C09077=1065.383,91.013,-73.073,172.465,27.858,155.108
C09078=1065.389,91.262,-73.092,172.466,27.861,155.108
C09079=1065.395,91.512,-73.110,172.467,27.864,155.108
C09080=1065.401,91.761,-73.128,172.469,27.867,155.109
C09081=1065.406,92.011,-73.147,172.470,27.869,155.109
C09082=1065.413,92.260,-73.165,172.472,27.872,155.110
C09083=1065.418,92.508,-73.184,172.474,27.875,155.110
C09084=1065.424,92.758,-73.202,172.475,27.878,155.110
C09085=1065.430,93.008,-73.221,172.477,27.880,155.111
C09086=1065.436,93.257,-73.240,172.478,27.883,155.111
C09087=1065.442,93.506,-73.258,172.480,27.886,155.112
C09088=1065.447,93.755,-73.277,172.481,27.889,155.112
C09089=1065.454,94.004,-73.295,172.483,27.892,155.112
C09090=1065.460,94.288,-73.316,172.484,27.894,155.113
C09091=1065.466,94.572,-73.338,172.486,27.898,155.113
C09092=1065.473,94.855,-73.358,172.488,27.901,155.114
C09093=1065.480,95.138,-73.380,172.490,27.904,155.114
C09094=1065.486,95.389,-73.399,172.491,27.906,155.114
C09095=1065.492,95.638,-73.417,172.493,27.909,155.115
C09096=1065.498,95.886,-73.436,172.494,27.912,155.115
C09097=1065.503,96.135,-73.455,172.496,27.915,155.116
C09098=1065.510,96.385,-73.473,172.497,27.918,155.116
C09099=1065.515,96.635,-73.492,172.499,27.920,155.116
C09100=1065.521,96.883,-73.510,172.501,27.923,155.117
C09101=1065.527,97.133,-73.529,172.501,27.926,155.117
C09102=1065.533,97.382,-73.548,172.503,27.928,155.118
C09103=1065.539,97.632,-73.567,172.504,27.931,155.118
C09104=1065.545,97.881,-73.585,172.506,27.933,155.118
C09105=1065.550,98.130,-73.604,172.507,27.936,155.119
C09106=1065.557,98.379,-73.623,172.509,27.939,155.119
C09107=1065.562,98.628,-73.642,172.510,27.942,155.120
C09108=1065.569,98.877,-73.661,172.512,27.945,155.120
C09109=1065.574,99.127,-73.680,172.514,27.947,155.120
C09110=1065.580,99.376,-73.698,172.515,27.950,155.121
C09111=1065.586,99.625,-73.717,172.517,27.953,155.121
C09112=1065.592,99.874,-73.735,172.518,27.955,155.121
C09113=1065.598,100.124,-73.755,172.520,27.958,155.122
C09114=1065.604,100.373,-73.773,172.521,27.961,155.122
C09115=1065.610,100.622,-73.793,172.523,27.963,155.123
C09116=1065.616,100.871,-73.811,172.524,27.966,155.123
C09117=1065.621,101.120,-73.830,172.526,27.969,155.123
C09118=1065.628,101.369,-73.849,172.528,27.972,155.124
C09119=1065.633,101.619,-73.868,172.529,27.975,155.124
C09120=1065.639,101.868,-73.887,172.531,27.977,155.125
C09121=1065.645,102.116,-73.905,172.532,27.980,155.125
C09122=1065.651,102.366,-73.925,172.534,27.983,155.125
C09123=1065.656,102.615,-73.944,172.535,27.986,155.126
C09124=1065.663,102.864,-73.963,172.537,27.988,155.126
C09125=1065.668,103.114,-73.982,172.538,27.991,155.127
C09126=1065.673,103.363,-74.001,172.540,27.994,155.127
C09127=1065.679,103.612,-74.020,172.542,27.996,155.127
C09128=1065.686,103.861,-74.039,172.543,27.999,155.128
C09129=1065.691,104.111,-74.058,172.545,28.002,155.128
C09130=1065.697,104.360,-74.077,172.546,28.005,155.129
C09131=1065.703,104.610,-74.096,172.548,28.007,155.129
C09132=1065.709,104.859,-74.115,172.549,28.010,155.129
C09133=1065.714,105.107,-74.134,172.551,28.013,155.130
C09134=1065.720,105.357,-74.153,172.552,28.016,155.130
C09135=1065.726,105.606,-74.172,172.554,28.018,155.131
C09136=1065.732,105.855,-74.191,172.556,28.021,155.131
C09137=1065.738,106.105,-74.210,172.557,28.024,155.131
C09138=1065.744,106.354,-74.230,172.559,28.027,155.132
C09139=1065.750,106.603,-74.249,172.560,28.030,155.132
C09140=1065.756,106.852,-74.268,172.562,28.032,155.133
C09141=1065.761,107.101,-74.287,172.563,28.035,155.133
C09142=1065.767,107.350,-74.306,172.565,28.037,155.133
C09143=1065.773,107.599,-74.325,172.567,28.040,155.134
C09144=1065.779,107.849,-74.344,172.568,28.043,155.134
C09145=1065.785,108.098,-74.364,172.570,28.046,155.134
C09146=1065.790,108.347,-74.383,172.571,28.048,155.135
C09147=1065.797,108.596,-74.402,172.573,28.051,155.135
C09148=1065.802,108.846,-74.421,172.574,28.054,155.136
C09149=1065.808,109.095,-74.440,172.576,28.057,155.136
C09150=1065.814,109.344,-74.460,172.577,28.060,155.136
C09151=1065.820,109.593,-74.480,172.579,28.062,155.137
C09152=1065.826,109.842,-74.498,172.581,28.064,155.137
C09153=1065.832,110.092,-74.518,172.582,28.067,155.138
C09154=1065.838,110.376,-74.540,172.584,28.071,155.138
C09155=1065.846,110.659,-74.562,172.585,28.073,155.138
C09156=1065.852,110.943,-74.584,172.587,28.077,155.139
C09157=1065.859,111.226,-74.606,172.589,28.080,155.139
C09158=1065.865,111.476,-74.626,172.591,28.083,155.140
C09159=1065.870,111.724,-74.644,172.592,28.085,155.140
C09160=1065.875,111.974,-74.664,172.594,28.088,155.141
C09161=1065.882,112.222,-74.683,172.595,28.091,155.141
C09162=1065.888,112.472,-74.702,172.597,28.094,155.141
C09163=1065.893,112.721,-74.721,172.598,28.096,155.142
C09164=1065.899,112.970,-74.741,172.600,28.099,155.142
C09165=1065.905,113.219,-74.761,172.602,28.102,155.143
C09166=1065.911,113.468,-74.781,172.603,28.104,155.143
C09167=1065.917,113.718,-74.800,172.605,28.107,155.143
C09168=1065.922,113.967,-74.819,172.606,28.110,155.144
C09169=1065.928,114.216,-74.839,172.608,28.112,155.144
C09170=1065.934,114.465,-74.858,172.609,28.115,155.145
C09171=1065.940,114.714,-74.878,172.611,28.118,155.145
C09172=1065.946,114.964,-74.898,172.613,28.121,155.145
C09173=1065.952,115.213,-74.917,172.614,28.124,155.146
C09174=1065.957,115.462,-74.937,172.616,28.126,155.146
C09175=1065.962,115.712,-74.957,172.617,28.129,155.147
C09176=1065.968,115.960,-74.977,172.619,28.132,155.147
C09177=1065.974,116.210,-74.996,172.620,28.135,155.147
C09178=1065.980,116.459,-75.016,172.622,28.137,155.148
C09179=1065.986,116.708,-75.035,172.624,28.140,155.148
C09180=1065.992,116.957,-75.055,172.625,28.143,155.149
C09181=1065.997,117.207,-75.075,172.627,28.146,155.149
C09182=1066.003,117.455,-75.095,172.628,28.149,155.149
C09183=1066.008,117.705,-75.114,172.630,28.152,155.150
C09184=1066.014,117.954,-75.134,172.631,28.155,155.150
C09185=1066.020,118.203,-75.153,172.633,28.157,155.151
C09186=1066.026,118.452,-75.173,172.634,28.160,155.151
C09187=1066.031,118.701,-75.194,172.636,28.163,155.151
C09188=1066.037,118.950,-75.213,172.638,28.166,155.152
C09189=1066.043,119.199,-75.233,172.639,28.168,155.152
C09190=1066.049,119.449,-75.252,172.641,28.171,155.153
C09191=1066.055,119.698,-75.272,172.642,28.173,155.153
C09192=1066.060,119.947,-75.293,172.644,28.176,155.153
C09193=1066.066,120.196,-75.312,172.646,28.179,155.154
C09194=1066.072,120.445,-75.332,172.648,28.182,155.154
C09195=1066.077,120.694,-75.351,172.650,28.185,155.155
C09196=1066.083,120.943,-75.371,172.651,28.187,155.155
C09197=1066.089,121.192,-75.392,172.653,28.190,155.155
C09198=1066.095,121.442,-75.411,172.654,28.193,155.156
C09199=1066.101,121.691,-75.431,172.656,28.196,155.156
C09200=1066.107,121.940,-75.451,172.657,28.198,155.157
C09201=1066.113,122.189,-75.470,172.659,28.201,155.157
C09202=1066.118,122.439,-75.491,172.660,28.204,155.157
C09203=1066.124,122.687,-75.511,172.662,28.207,155.158
C09204=1066.130,122.937,-75.530,172.664,28.209,155.158
C09205=1066.136,123.186,-75.550,172.665,28.212,155.159
C09206=1066.142,123.434,-75.570,172.667,28.215,155.159
C09207=1066.147,123.684,-75.591,172.668,28.218,155.159
C09208=1066.153,123.934,-75.610,172.670,28.221,155.160
C09209=1066.159,124.183,-75.630,172.671,28.223,155.160
C09210=1066.165,124.431,-75.650,172.673,28.226,155.161
C09211=1066.170,124.680,-75.671,172.675,28.229,155.161
C09212=1066.176,124.930,-75.690,172.677,28.232,155.161
C09213=1066.182,125.179,-75.710,172.679,28.234,155.162
C09214=1066.188,125.428,-75.730,172.680,28.237,155.162
C09215=1066.194,125.677,-75.751,172.682,28.240,155.162
C09216=1066.200,125.926,-75.771,172.683,28.242,155.163
C09217=1066.206,126.175,-75.791,172.685,28.245,155.163
C09218=1066.212,126.459,-75.813,172.687,28.248,155.164
C09219=1066.218,126.743,-75.836,172.689,28.251,155.164
C09220=1066.226,127.026,-75.859,172.691,28.255,155.165
C09221=1066.232,127.310,-75.882,172.692,28.257,155.165
C09222=1066.238,127.559,-75.902,172.694,28.260,155.166
C09223=1066.244,127.808,-75.922,172.695,28.263,155.166
C09224=1066.249,128.057,-75.942,172.698,28.266,155.166
C09225=1066.256,128.306,-75.962,172.699,28.269,155.167
C09226=1066.262,128.555,-75.982,172.701,28.271,155.167
C09227=1066.267,128.804,-76.003,172.703,28.274,155.167
C09228=1066.273,129.053,-76.023,172.704,28.276,155.168
C09229=1066.280,129.303,-76.043,172.706,28.279,155.168
C09230=1066.286,129.551,-76.063,172.707,28.282,155.169
C09231=1066.291,129.800,-76.084,172.709,28.285,155.169
C09232=1066.297,130.050,-76.103,172.710,28.287,155.169
C09233=1066.303,130.299,-76.123,172.712,28.290,155.170
C09234=1066.309,130.549,-76.144,172.714,28.292,155.170
C09235=1066.315,130.797,-76.164,172.716,28.295,155.171
C09236=1066.321,131.046,-76.184,172.718,28.298,155.171
C09237=1066.327,131.296,-76.205,172.719,28.301,155.171
C09238=1066.333,131.545,-76.225,172.721,28.304,155.172
C09239=1066.339,131.794,-76.245,172.723,28.306,155.172
C09240=1066.344,132.043,-76.266,172.724,28.309,155.173
C09241=1066.351,132.292,-76.286,172.726,28.312,155.173
C09242=1066.356,132.541,-76.307,172.727,28.315,155.173
C09243=1066.362,132.790,-76.327,172.729,28.317,155.174
C09244=1066.367,133.039,-76.347,172.730,28.320,155.174
C09245=1066.374,133.288,-76.368,172.733,28.323,155.175
C09246=1066.379,133.537,-76.388,172.735,28.326,155.175
C09247=1066.384,133.786,-76.409,172.736,28.329,155.175
C09248=1066.390,134.035,-76.429,172.738,28.331,155.176
C09249=1066.396,134.285,-76.450,172.739,28.334,155.176
C09250=1066.402,134.534,-76.470,172.741,28.337,155.177
C09251=1066.408,134.782,-76.491,172.742,28.340,155.177
C09252=1066.414,135.031,-76.511,172.744,28.342,155.177
C09253=1066.420,135.281,-76.532,172.746,28.345,155.178
C09254=1066.425,135.530,-76.552,172.747,28.348,155.178
C09255=1066.431,135.779,-76.572,172.750,28.350,155.178
C09256=1066.437,136.029,-76.593,172.751,28.353,155.179
C09257=1066.443,136.277,-76.614,172.753,28.356,155.179
C09258=1066.448,136.526,-76.634,172.755,28.359,155.180
C09259=1066.454,136.776,-76.655,172.756,28.361,155.180
C09260=1066.460,137.025,-76.675,172.758,28.364,155.180
C09261=1066.466,137.273,-76.697,172.759,28.367,155.181
C09262=1066.472,137.523,-76.717,172.761,28.370,155.181
C09263=1066.477,137.772,-76.737,172.763,28.373,155.182
C09264=1066.483,138.021,-76.758,172.765,28.375,155.182
C09265=1066.490,138.270,-76.779,172.767,28.378,155.182
C09266=1066.495,138.519,-76.800,172.768,28.381,155.183
C09267=1066.500,138.768,-76.820,172.770,28.384,155.183
C09268=1066.507,139.018,-76.840,172.771,28.386,155.184
C09269=1066.512,139.266,-76.862,172.773,28.389,155.184
C09270=1066.518,139.515,-76.882,172.775,28.392,155.184
C09271=1066.524,139.765,-76.903,172.777,28.395,155.185
C09272=1066.530,140.013,-76.924,172.779,28.398,155.185
C09273=1066.535,140.262,-76.944,172.780,28.400,155.186
C09274=1066.542,140.512,-76.965,172.782,28.403,155.186
C09275=1066.547,140.760,-76.986,172.783,28.406,155.187
C09276=1066.552,141.010,-77.007,172.785,28.409,155.187
C09277=1066.559,141.259,-77.028,172.788,28.411,155.187
C09278=1066.564,141.508,-77.049,172.789,28.414,155.188
C09279=1066.570,141.757,-77.069,172.791,28.417,155.188
C09280=1066.576,142.006,-77.090,172.792,28.420,155.189
C09281=1066.581,142.255,-77.111,172.794,28.422,155.189
C09282=1066.588,142.539,-77.135,172.796,28.426,155.189
C09283=1066.594,142.822,-77.159,172.798,28.429,155.190
C09284=1066.600,143.105,-77.183,172.799,28.432,155.190
C09285=1066.608,143.389,-77.206,172.802,28.435,155.191
C09286=1066.613,143.638,-77.227,172.804,28.438,155.191
C09287=1066.619,143.887,-77.249,172.805,28.441,155.192
C09288=1066.625,144.136,-77.269,172.807,28.443,155.192
C09289=1066.630,144.385,-77.290,172.809,28.446,155.192
C09290=1066.636,144.635,-77.311,172.811,28.449,155.193
C09291=1066.642,144.883,-77.332,172.812,28.452,155.193
C09292=1066.648,145.132,-77.354,172.814,28.454,155.194
C09293=1066.654,145.381,-77.374,172.816,28.457,155.194
C09294=1066.660,145.630,-77.396,172.817,28.460,155.194
C09295=1066.665,145.880,-77.416,172.820,28.463,155.195
C09296=1066.671,146.128,-77.438,172.821,28.466,155.195
C09297=1066.677,146.378,-77.458,172.823,28.468,155.196
C09298=1066.683,146.626,-77.479,172.825,28.471,155.196
C09299=1066.689,146.875,-77.501,172.826,28.474,155.196
C09300=1066.694,147.124,-77.521,172.828,28.477,155.197
C09301=1066.700,147.374,-77.543,172.830,28.480,155.197
C09302=1066.706,147.623,-77.564,172.832,28.482,155.198
C09303=1066.712,147.872,-77.585,172.833,28.485,155.198
C09304=1066.717,148.120,-77.606,172.835,28.488,155.198
C09305=1066.723,148.370,-77.627,172.837,28.491,155.199
C09306=1066.729,148.619,-77.649,172.839,28.494,155.199
C09307=1066.735,148.868,-77.670,172.841,28.496,155.200
C09308=1066.740,149.117,-77.691,172.842,28.499,155.200
C09309=1066.746,149.366,-77.712,172.844,28.502,155.200
C09310=1066.752,149.615,-77.734,172.846,28.504,155.201
C09311=1066.758,149.864,-77.755,172.847,28.507,155.201
C09312=1066.763,150.113,-77.776,172.850,28.510,155.202
C09313=1066.769,150.362,-77.797,172.851,28.513,155.202
C09314=1066.775,150.611,-77.819,172.853,28.516,155.202
C09315=1066.780,150.860,-77.839,172.855,28.518,155.203
C09316=1066.787,151.109,-77.861,172.856,28.521,155.203
C09317=1066.792,151.358,-77.882,172.859,28.524,155.204
C09318=1066.798,151.607,-77.904,172.860,28.527,155.204
C09319=1066.804,151.856,-77.926,172.862,28.530,155.204
C09320=1066.809,152.106,-77.947,172.863,28.532,155.205
C09321=1066.815,152.355,-77.968,172.866,28.536,155.205
C09322=1066.821,152.603,-77.990,172.868,28.539,155.206
C09323=1066.827,152.852,-78.011,172.869,28.541,155.206
C09324=1066.832,153.101,-78.033,172.871,28.544,155.207
C09325=1066.839,153.350,-78.054,172.872,28.547,155.207
C09326=1066.844,153.599,-78.075,172.875,28.550,155.207
C09327=1066.850,153.848,-78.096,172.876,28.552,155.208
C09328=1066.856,154.097,-78.118,172.878,28.555,155.208
C09329=1066.861,154.346,-78.140,172.880,28.558,155.209
C09330=1066.867,154.596,-78.161,172.881,28.561,155.209
C09331=1066.873,154.844,-78.183,172.884,28.564,155.209
C09332=1066.879,155.093,-78.204,172.885,28.566,155.210
C09333=1066.884,155.342,-78.226,172.887,28.569,155.210
C09334=1066.891,155.591,-78.247,172.889,28.572,155.211
C09335=1066.895,155.840,-78.269,172.891,28.575,155.211
C09336=1066.902,156.089,-78.291,172.893,28.578,155.211
C09337=1066.908,156.338,-78.312,172.894,28.580,155.212
C09338=1066.913,156.587,-78.334,172.896,28.583,155.212
C09339=1066.919,156.836,-78.356,172.899,28.586,155.213
C09340=1066.924,157.085,-78.377,172.900,28.589,155.213
C09341=1066.930,157.334,-78.399,172.902,28.591,155.213
C09342=1066.937,157.583,-78.420,172.903,28.594,155.214
C09343=1066.941,157.832,-78.442,172.906,28.598,155.214
C09344=1066.948,158.081,-78.464,172.907,28.600,155.215
C09345=1066.953,158.330,-78.485,172.909,28.603,155.215
C09346=1066.960,158.613,-78.510,172.912,28.606,155.215
C09347=1066.966,158.896,-78.535,172.913,28.609,155.216
C09348=1066.973,159.180,-78.560,172.916,28.612,155.216
C09349=1066.980,159.463,-78.584,172.917,28.616,155.217
C09350=1066.985,159.712,-78.606,172.920,28.619,155.217
C09351=1066.991,159.961,-78.628,172.921,28.621,155.218
C09352=1066.996,160.210,-78.649,172.923,28.624,155.218
C09353=1067.003,160.459,-78.671,172.925,28.627,155.219
C09354=1067.008,160.708,-78.693,172.927,28.630,155.219
C09355=1067.015,160.957,-78.715,172.929,28.632,155.219
C09356=1067.020,161.205,-78.737,172.930,28.635,155.220
C09357=1067.026,161.455,-78.759,172.932,28.638,155.220
C09358=1067.031,161.703,-78.780,172.935,28.641,155.221
C09359=1067.036,161.953,-78.802,172.936,28.644,155.221
C09360=1067.042,162.202,-78.825,172.938,28.647,155.221
C09361=1067.048,162.450,-78.847,172.939,28.650,155.222
C09362=1067.053,162.700,-78.869,172.942,28.653,155.222
C09363=1067.059,162.948,-78.890,172.943,28.656,155.223
C09364=1067.065,163.197,-78.913,172.945,28.659,155.223
C09365=1067.070,163.447,-78.935,172.948,28.662,155.224
C09366=1067.075,163.695,-78.956,172.949,28.665,155.224
C09367=1067.081,163.945,-78.979,172.951,28.668,155.224
C09368=1067.087,164.193,-79.001,172.952,28.670,155.225
C09369=1067.092,164.442,-79.023,172.955,28.673,155.225
C09370=1067.098,164.692,-79.045,172.956,28.677,155.226
C09371=1067.103,164.940,-79.067,172.958,28.679,155.226
C09372=1067.109,165.189,-79.089,172.961,28.682,155.227
C09373=1067.114,165.439,-79.112,172.962,28.685,155.227
C09374=1067.120,165.687,-79.134,172.964,28.688,155.227
C09375=1067.126,165.936,-79.156,172.965,28.691,155.228
C09376=1067.131,166.186,-79.178,172.968,28.694,155.228
C09377=1067.138,166.434,-79.200,172.970,28.697,155.229
C09378=1067.142,166.683,-79.222,172.971,28.699,155.229
C09379=1067.148,166.932,-79.245,172.974,28.702,155.230
C09380=1067.154,167.181,-79.267,172.975,28.706,155.230
C09381=1067.159,167.429,-79.289,172.977,28.708,155.230
C09382=1067.165,167.679,-79.312,172.979,28.711,155.231
C09383=1067.171,167.928,-79.333,172.981,28.714,155.231
C09384=1067.177,168.177,-79.356,172.983,28.717,155.232
C09385=1067.182,168.426,-79.378,172.984,28.720,155.232
C09386=1067.188,168.674,-79.400,172.987,28.723,155.233
C09387=1067.193,168.924,-79.423,172.988,28.726,155.233
C09388=1067.199,169.172,-79.445,172.990,28.728,155.233
C09389=1067.205,169.421,-79.467,172.993,28.731,155.234
C09390=1067.210,169.670,-79.490,172.994,28.735,155.234
C09391=1067.216,169.920,-79.512,172.996,28.737,155.235
C09392=1067.222,170.168,-79.534,172.998,28.740,155.235
C09393=1067.227,170.417,-79.556,173.000,28.743,155.236
C09394=1067.233,170.666,-79.579,173.002,28.746,155.236
C09395=1067.239,170.915,-79.602,173.004,28.749,155.236
C09396=1067.245,171.164,-79.624,173.006,28.752,155.237
C09397=1067.251,171.413,-79.647,173.007,28.755,155.237
C09398=1067.255,171.662,-79.669,173.010,28.758,155.238
C09399=1067.262,171.910,-79.691,173.012,28.760,155.238
C09400=1067.268,172.159,-79.714,173.013,28.763,155.238
C09401=1067.273,172.409,-79.736,173.016,28.766,155.239
C09402=1067.279,172.658,-79.759,173.017,28.769,155.239
C09403=1067.285,172.906,-79.781,173.019,28.772,155.240
C09404=1067.290,173.155,-79.803,173.021,28.775,155.240
C09405=1067.296,173.404,-79.826,173.023,28.778,155.241
C09406=1067.301,173.653,-79.849,173.025,28.780,155.241
C09407=1067.308,173.902,-79.871,173.027,28.784,155.242
C09408=1067.313,174.151,-79.894,173.029,28.786,155.242
C09409=1067.319,174.400,-79.917,173.031,28.789,155.242
C09410=1067.325,174.683,-79.941,173.033,28.793,155.243
C09411=1067.332,174.966,-79.967,173.036,28.796,155.243
C09412=1067.338,175.248,-79.993,173.038,28.799,155.244
C09413=1067.345,175.531,-80.019,173.040,28.802,155.244
C09414=1067.351,175.780,-80.041,173.042,28.805,155.245
C09415=1067.357,176.029,-80.064,173.044,28.808,155.245
C09416=1067.363,176.278,-80.087,173.045,28.811,155.245
C09417=1067.368,176.527,-80.109,173.048,28.814,155.246
C09418=1067.374,176.776,-80.132,173.050,28.817,155.246
C09419=1067.380,177.025,-80.155,173.052,28.820,155.247
C09420=1067.386,177.273,-80.178,173.054,28.823,155.247
C09421=1067.392,177.522,-80.200,173.055,28.825,155.248
C09422=1067.397,177.772,-80.223,173.058,28.828,155.248
C09423=1067.403,178.020,-80.245,173.060,28.831,155.248
C09424=1067.409,178.269,-80.268,173.062,28.835,155.249
C09425=1067.414,178.518,-80.291,173.064,28.837,155.249
C09426=1067.420,178.766,-80.313,173.065,28.840,155.250
C09427=1067.426,179.015,-80.336,173.068,28.843,155.250
C09428=1067.432,179.264,-80.359,173.070,28.846,155.251
C09429=1067.438,179.513,-80.382,173.072,28.849,155.251
C09430=1067.444,179.762,-80.405,173.074,28.851,155.251
C09431=1067.450,180.011,-80.428,173.075,28.854,155.252
C09432=1067.455,180.260,-80.450,173.078,28.857,155.252
C09433=1067.461,180.509,-80.473,173.080,28.860,155.253
C09434=1067.467,180.758,-80.495,173.082,28.863,155.253
C09435=1067.473,181.006,-80.518,173.084,28.866,155.253
C09436=1067.479,181.256,-80.541,173.086,28.869,155.254
C09437=1067.485,181.505,-80.564,173.088,28.871,155.254
C09438=1067.491,181.754,-80.587,173.090,28.875,155.255
C09439=1067.496,182.003,-80.610,173.092,28.878,155.255
C09440=1067.503,182.251,-80.633,173.094,28.880,155.256
C09441=1067.509,182.500,-80.656,173.096,28.883,155.256
C09442=1067.514,182.749,-80.678,173.098,28.886,155.256
C09443=1067.520,182.997,-80.702,173.101,28.889,155.257
C09444=1067.526,183.246,-80.725,173.102,28.892,155.257
C09445=1067.532,183.495,-80.748,173.104,28.894,155.258
C09446=1067.538,183.744,-80.771,173.106,28.898,155.258
C09447=1067.544,183.993,-80.793,173.108,28.900,155.258
C09448=1067.550,184.242,-80.816,173.111,28.903,155.259
C09449=1067.556,184.491,-80.840,173.112,28.906,155.259
C09450=1067.562,184.740,-80.863,173.115,28.909,155.260
C09451=1067.568,184.989,-80.885,173.116,28.912,155.260
C09452=1067.573,185.238,-80.910,173.119,28.915,155.261
C09453=1067.579,185.486,-80.933,173.121,28.918,155.261
C09454=1067.584,185.735,-80.956,173.122,28.921,155.262
C09455=1067.589,185.985,-80.979,173.125,28.924,155.262
C09456=1067.595,186.233,-81.002,173.126,28.927,155.262
C09457=1067.601,186.482,-81.026,173.129,28.930,155.263
C09458=1067.606,186.731,-81.049,173.130,28.933,155.263
C09459=1067.612,186.980,-81.072,173.133,28.936,155.264
C09460=1067.618,187.229,-81.095,173.135,28.939,155.264
C09461=1067.623,187.477,-81.119,173.137,28.943,155.265
C09462=1067.629,187.726,-81.142,173.139,28.945,155.265
C09463=1067.634,187.975,-81.165,173.141,28.949,155.266
C09464=1067.640,188.224,-81.190,173.143,28.952,155.266
C09465=1067.645,188.473,-81.213,173.146,28.954,155.266
C09466=1067.651,188.722,-81.236,173.147,28.958,155.267
C09467=1067.656,188.970,-81.260,173.149,28.960,155.267
C09468=1067.662,189.219,-81.283,173.151,28.964,155.268
C09469=1067.668,189.468,-81.306,173.153,28.967,155.268
C09470=1067.673,189.716,-81.330,173.156,28.970,155.269
C09471=1067.679,189.965,-81.353,173.157,28.973,155.269
C09472=1067.685,190.215,-81.376,173.160,28.976,155.270
C09473=1067.691,190.464,-81.400,173.161,28.979,155.270
C09474=1067.697,190.745,-81.427,173.164,28.982,155.271
C09475=1067.704,191.028,-81.454,173.166,28.986,155.271
C09476=1067.710,191.311,-81.480,173.169,28.989,155.272
C09477=1067.716,191.593,-81.507,173.171,28.993,155.272
C09478=1067.722,191.841,-81.530,173.173,28.996,155.273
C09479=1067.728,192.091,-81.554,173.176,28.998,155.273
C09480=1067.734,192.340,-81.578,173.177,29.002,155.273
C09481=1067.739,192.588,-81.601,173.180,29.005,155.274
C09482=1067.745,192.837,-81.625,173.181,29.008,155.274
C09483=1067.750,193.086,-81.648,173.184,29.011,155.275
C09484=1067.756,193.334,-81.672,173.186,29.014,155.275
C09485=1067.762,193.584,-81.696,173.188,29.017,155.276
C09486=1067.768,193.832,-81.719,173.190,29.020,155.276
C09487=1067.773,194.081,-81.743,173.192,29.023,155.277
C09488=1067.779,194.330,-81.766,173.194,29.026,155.277
C09489=1067.784,194.578,-81.791,173.196,29.029,155.278
C09490=1067.791,194.828,-81.814,173.198,29.032,155.278
C09491=1067.797,195.076,-81.838,173.201,29.035,155.278
C09492=1067.802,195.325,-81.862,173.202,29.038,155.279
C09493=1067.808,195.574,-81.885,173.205,29.041,155.279
C09494=1067.814,195.823,-81.909,173.207,29.045,155.280
C09495=1067.819,196.072,-81.932,173.209,29.047,155.280
C09496=1067.825,196.321,-81.957,173.212,29.050,155.281
C09497=1067.831,196.569,-81.980,173.213,29.053,155.281
C09498=1067.837,196.818,-82.004,173.216,29.056,155.281
C09499=1067.842,197.067,-82.028,173.217,29.060,155.282
C09500=1067.848,197.315,-82.052,173.220,29.062,155.282
C09501=1067.854,197.564,-82.076,173.222,29.066,155.283
C09502=1067.860,197.813,-82.099,173.224,29.069,155.283
C09503=1067.865,198.062,-82.123,173.227,29.072,155.284
C09504=1067.871,198.310,-82.147,173.228,29.075,155.284
C09505=1067.877,198.560,-82.172,173.231,29.078,155.285
C09506=1067.883,198.809,-82.195,173.233,29.081,155.285
C09507=1067.888,199.057,-82.219,173.235,29.084,155.286
C09508=1067.895,199.306,-82.243,173.237,29.087,155.286
C09509=1067.901,199.554,-82.267,173.239,29.090,155.287
C09510=1067.906,199.803,-82.291,173.242,29.093,155.287
C09511=1067.913,200.053,-82.314,173.244,29.096,155.287
C09512=1067.918,200.301,-82.338,173.246,29.099,155.288
C09513=1067.924,200.549,-82.362,173.248,29.102,155.288
C09514=1067.930,200.799,-82.387,173.250,29.105,155.289
C09515=1067.936,201.047,-82.410,173.252,29.108,155.289
C09516=1067.941,201.296,-82.435,173.255,29.111,155.290
C09517=1067.948,201.545,-82.459,173.257,29.114,155.290
C09518=1067.953,201.794,-82.482,173.259,29.118,155.291
C09519=1067.959,202.043,-82.506,173.261,29.120,155.291
C09520=1067.965,202.291,-82.530,173.263,29.124,155.292
C09521=1067.970,202.540,-82.555,173.266,29.127,155.292
C09522=1067.977,202.789,-82.579,173.268,29.130,155.292
C09523=1067.982,203.037,-82.603,173.270,29.133,155.293
C09524=1067.987,203.286,-82.627,173.272,29.136,155.293
C09525=1067.993,203.535,-82.652,173.274,29.139,155.294
C09526=1067.998,203.784,-82.676,173.277,29.142,155.294
C09527=1068.004,204.032,-82.700,173.279,29.146,155.295
C09528=1068.010,204.282,-82.724,173.281,29.148,155.295
C09529=1068.016,204.530,-82.749,173.283,29.152,155.296
C09530=1068.022,204.779,-82.773,173.286,29.155,155.296
C09531=1068.028,205.028,-82.797,173.287,29.158,155.297
C09532=1068.033,205.276,-82.821,173.290,29.162,155.297
C09533=1068.039,205.525,-82.846,173.292,29.164,155.298
C09534=1068.044,205.773,-82.871,173.294,29.168,155.298
C09535=1068.050,206.023,-82.895,173.297,29.171,155.299
C09536=1068.056,206.271,-82.919,173.298,29.174,155.299
C09537=1068.062,206.520,-82.943,173.301,29.177,155.300
C09538=1068.086,207.564,-83.046,173.447,29.251,155.303
C09539=1068.092,207.797,-83.070,173.450,29.255,155.304
C09540=1068.097,208.030,-83.093,173.451,29.259,155.305
C09541=1068.103,208.263,-83.117,173.453,29.263,155.305
C09542=1068.108,208.496,-83.140,173.455,29.267,155.306
C09543=1068.114,208.728,-83.164,173.457,29.270,155.307
C09544=1068.119,208.962,-83.188,173.458,29.274,155.307
C09545=1068.125,209.194,-83.211,173.461,29.278,155.308
C09546=1068.130,209.427,-83.234,173.462,29.282,155.308
C09547=1068.136,209.676,-83.260,173.465,29.286,155.309
C09548=1068.142,209.924,-83.285,173.466,29.290,155.310
C09549=1068.148,210.173,-83.311,173.469,29.294,155.311
C09550=1068.155,210.422,-83.336,173.470,29.298,155.311
C09551=1068.160,210.670,-83.360,173.473,29.302,155.312
C09552=1068.166,210.919,-83.386,173.474,29.306,155.313
C09553=1068.171,211.168,-83.412,173.477,29.310,155.313
C09554=1068.178,211.417,-83.437,173.478,29.314,155.314
C09555=1068.184,211.665,-83.462,173.481,29.319,155.315
C09556=1068.189,211.913,-83.487,173.482,29.322,155.315
C09557=1068.195,212.162,-83.513,173.485,29.326,155.316
C09558=1068.201,212.411,-83.538,173.486,29.331,155.317
C09559=1068.207,212.660,-83.564,173.489,29.335,155.317
C09560=1068.214,212.908,-83.589,173.490,29.338,155.318
C09561=1068.219,213.157,-83.615,173.493,29.342,155.319
C09562=1068.225,213.405,-83.640,173.494,29.347,155.319
C09563=1068.231,213.654,-83.665,173.497,29.351,155.320
C09564=1068.236,213.903,-83.691,173.499,29.354,155.321
C09565=1068.243,214.152,-83.717,173.501,29.359,155.322
C09566=1068.249,214.400,-83.742,173.503,29.363,155.322
C09567=1068.254,214.649,-83.768,173.505,29.367,155.323
C09568=1068.260,214.898,-83.793,173.507,29.371,155.324
C09569=1068.266,215.146,-83.820,173.509,29.375,155.324
C09570=1068.272,215.394,-83.845,173.511,29.379,155.325
C09571=1068.278,215.643,-83.870,173.513,29.383,155.326
C09572=1068.283,215.892,-83.896,173.516,29.387,155.326
C09573=1068.290,216.141,-83.921,173.517,29.391,155.327
C09574=1068.295,216.390,-83.947,173.520,29.396,155.328
C09575=1068.301,216.638,-83.973,173.521,29.399,155.328
C09576=1068.308,216.886,-83.999,173.524,29.403,155.329
C09577=1068.313,217.135,-84.025,173.525,29.407,155.330
C09578=1068.319,217.383,-84.050,173.528,29.412,155.330
C09579=1068.324,217.616,-84.074,173.529,29.415,155.331
C09580=1068.330,217.847,-84.098,173.532,29.419,155.332
C09581=1068.335,218.080,-84.122,173.533,29.423,155.332
C09582=1068.341,218.311,-84.146,173.535,29.426,155.333
C09583=1068.347,218.543,-84.170,173.537,29.430,155.334
C09584=1068.352,218.776,-84.194,173.539,29.434,155.334
C09585=1068.358,219.007,-84.218,173.542,29.437,155.335
C09586=1068.363,219.239,-84.242,173.543,29.441,155.335
C09587=1068.370,219.487,-84.269,173.545,29.445,155.336
C09588=1068.375,219.736,-84.294,173.547,29.449,155.337
C09589=1068.381,219.985,-84.320,173.550,29.453,155.337
C09590=1068.388,220.233,-84.346,173.551,29.457,155.338
C09591=1068.393,220.482,-84.372,173.554,29.461,155.339
C09592=1068.399,220.730,-84.397,173.555,29.466,155.340
C09593=1068.405,220.979,-84.424,173.558,29.469,155.340
C09594=1068.411,221.227,-84.449,173.560,29.473,155.341
C09595=1068.416,221.446,-84.472,173.562,29.477,155.341
C09596=1068.422,221.664,-84.495,173.563,29.480,155.342
C09597=1068.427,221.883,-84.518,173.565,29.484,155.343
C09598=1068.432,222.101,-84.541,173.568,29.488,155.343
C09599=1068.437,222.320,-84.563,173.569,29.491,155.344
C09600=1068.442,222.539,-84.586,173.571,29.495,155.344
C09601=1068.447,222.756,-84.609,173.572,29.498,155.345
C09602=1068.452,222.974,-84.632,173.575,29.502,155.346
C09603=1068.458,223.223,-84.658,173.577,29.505,155.346
C09604=1068.464,223.472,-84.684,173.579,29.510,155.347
C09605=1068.469,223.720,-84.711,173.581,29.514,155.348
C09606=1068.476,223.970,-84.737,173.583,29.518,155.348
C09607=1068.482,224.218,-84.763,173.586,29.522,155.349
C09608=1068.488,224.466,-84.790,173.587,29.526,155.350
C09609=1068.494,224.715,-84.815,173.590,29.530,155.350
C09610=1068.500,224.963,-84.842,173.591,29.534,155.351
C09611=1068.505,225.212,-84.868,173.594,29.538,155.352
C09612=1068.512,225.460,-84.894,173.596,29.542,155.352
C09613=1068.517,225.709,-84.921,173.598,29.546,155.353
C09614=1068.523,225.958,-84.947,173.600,29.550,155.354
C09615=1068.529,226.206,-84.973,173.602,29.554,155.354
C09616=1068.535,226.455,-84.999,173.605,29.558,155.355
C09617=1068.541,226.703,-85.025,173.607,29.562,155.356
C09618=1068.546,226.951,-85.052,173.609,29.566,155.357
C09619=1068.553,227.200,-85.079,173.611,29.570,155.357
C09620=1068.559,227.449,-85.104,173.614,29.574,155.358
C09621=1068.565,227.698,-85.131,173.615,29.577,155.358
C09622=1068.571,227.946,-85.157,173.618,29.582,155.359
C09623=1068.576,228.195,-85.183,173.620,29.586,155.360
C09624=1068.583,228.443,-85.209,173.622,29.590,155.361
C09625=1068.589,228.692,-85.236,173.624,29.594,155.361
C09626=1068.595,228.940,-85.263,173.626,29.597,155.362
C09627=1068.601,229.189,-85.290,173.628,29.601,155.362
C09628=1068.607,229.437,-85.315,173.631,29.605,155.363
C09629=1068.612,229.686,-85.342,173.633,29.610,155.364
C09630=1068.619,229.935,-85.369,173.635,29.614,155.365
C09631=1068.625,230.183,-85.395,173.638,29.617,155.365
C09632=1068.630,230.431,-85.422,173.639,29.621,155.366
C09633=1068.636,230.680,-85.449,173.642,29.625,155.366
C09634=1068.642,230.929,-85.475,173.644,29.630,155.367
C09635=1068.647,231.177,-85.501,173.646,29.633,155.368
C09636=1068.654,231.426,-85.528,173.648,29.637,155.369
C09637=1068.660,231.675,-85.555,173.651,29.641,155.369
C09638=1068.665,231.923,-85.582,173.652,29.646,155.370
C09639=1068.671,232.171,-85.608,173.655,29.650,155.371
C09640=1068.677,232.420,-85.635,173.658,29.653,155.371
C09641=1068.683,232.669,-85.662,173.659,29.657,155.372
C09642=1068.689,232.917,-85.689,173.662,29.661,155.373
C09643=1068.695,233.165,-85.715,173.664,29.666,155.373
C09644=1068.701,233.414,-85.742,173.666,29.669,155.374
C09645=1068.706,233.662,-85.768,173.668,29.673,155.375
C09646=1068.713,233.911,-85.796,173.671,29.677,155.375
C09647=1068.719,234.160,-85.822,173.673,29.681,155.376
C09648=1068.724,234.408,-85.849,173.675,29.686,155.377
C09649=1068.730,234.656,-85.875,173.678,29.689,155.377
C09650=1068.736,234.905,-85.902,173.679,29.693,155.378
C09651=1068.741,235.120,-85.926,173.682,29.697,155.379
C09652=1068.746,235.334,-85.950,173.683,29.700,155.379
C09653=1068.752,235.548,-85.972,173.685,29.703,155.380
C09654=1068.757,235.762,-85.995,173.687,29.707,155.380
C09655=1068.761,235.976,-86.019,173.689,29.711,155.381
C09656=1068.766,236.191,-86.042,173.691,29.714,155.382
C09657=1068.772,236.405,-86.065,173.692,29.718,155.382
C09658=1068.777,236.620,-86.089,173.695,29.721,155.383
C09659=1068.783,236.868,-86.115,173.697,29.725,155.383
C09660=1068.789,237.117,-86.142,173.699,29.729,155.384
C09661=1068.795,237.365,-86.169,173.702,29.733,155.385
C09662=1068.800,237.614,-86.197,173.704,29.737,155.385
C09663=1068.806,237.862,-86.224,173.706,29.741,155.386
C09664=1068.812,238.110,-86.250,173.708,29.745,155.387
C09665=1068.818,238.359,-86.277,173.711,29.749,155.387
C09666=1068.824,238.607,-86.305,173.713,29.752,155.388
C09667=1068.830,238.856,-86.331,173.715,29.757,155.389
C09668=1068.836,239.105,-86.359,173.718,29.761,155.389
C09669=1068.842,239.353,-86.386,173.720,29.765,155.390
C09670=1068.848,239.602,-86.413,173.722,29.768,155.391
C09671=1068.854,239.850,-86.440,173.724,29.772,155.391
C09672=1068.860,240.098,-86.467,173.727,29.776,155.392
C09673=1068.866,240.347,-86.495,173.729,29.780,155.393
C09674=1068.872,240.596,-86.522,173.731,29.784,155.393
C09675=1068.878,240.843,-86.549,173.734,29.788,155.394
C09676=1068.884,241.092,-86.576,173.736,29.792,155.395
C09677=1068.889,241.340,-86.604,173.738,29.796,155.395
C09678=1068.896,241.590,-86.631,173.740,29.800,155.396
C09679=1068.902,241.837,-86.658,173.743,29.804,155.397
C09680=1068.908,242.086,-86.685,173.746,29.808,155.397
C09681=1068.913,242.335,-86.713,173.747,29.812,155.398
C09682=1068.919,242.583,-86.740,173.750,29.816,155.399
C09683=1068.926,242.832,-86.767,173.752,29.820,155.399
C09684=1068.931,243.080,-86.795,173.755,29.824,155.400
C09685=1068.938,243.328,-86.823,173.756,29.828,155.401
C09686=1068.943,243.577,-86.850,173.759,29.832,155.402
C09687=1068.949,243.825,-86.877,173.762,29.836,155.402
C09688=1068.954,244.074,-86.905,173.764,29.840,155.403
C09689=1068.961,244.322,-86.932,173.766,29.844,155.404
C09690=1068.967,244.571,-86.959,173.768,29.848,155.404
C09691=1068.972,244.819,-86.987,173.771,29.852,155.405
C09692=1068.979,245.067,-87.015,173.773,29.856,155.406
C09693=1068.984,245.316,-87.042,173.775,29.860,155.406
C09694=1068.990,245.564,-87.070,173.778,29.864,155.407
C09695=1068.996,245.813,-87.098,173.780,29.868,155.408
C09696=1069.002,246.061,-87.124,173.783,29.872,155.408
C09697=1069.008,246.310,-87.153,173.784,29.876,155.409
C09698=1069.014,246.557,-87.180,173.787,29.880,155.410
C09699=1069.019,246.807,-87.208,173.790,29.884,155.410
C09700=1069.026,247.054,-87.235,173.792,29.888,155.411
C09701=1069.031,247.303,-87.263,173.794,29.892,155.412
C09702=1069.037,247.551,-87.291,173.796,29.896,155.412
C09703=1069.043,247.800,-87.318,173.799,29.900,155.413
C09704=1069.049,248.048,-87.346,173.801,29.904,155.414
C09705=1069.054,248.297,-87.375,173.804,29.908,155.414
C09706=1069.061,248.545,-87.402,173.806,29.912,155.415
C09707=1069.065,248.756,-87.426,173.808,29.916,155.416
C09708=1069.070,248.967,-87.450,173.810,29.919,155.416
C09709=1069.075,249.179,-87.474,173.812,29.922,155.417
C09710=1069.080,249.390,-87.497,173.814,29.926,155.417
C09711=1069.085,249.601,-87.521,173.816,29.929,155.418
C09712=1069.090,249.812,-87.545,173.818,29.932,155.419
C09713=1069.095,250.023,-87.568,173.820,29.936,155.419
C09714=1069.100,250.234,-87.592,173.822,29.939,155.420
C09715=1069.106,250.482,-87.620,173.824,29.943,155.420
C09716=1069.112,250.731,-87.648,173.827,29.947,155.421
C09717=1069.118,250.979,-87.676,173.829,29.951,155.422
C09718=1069.124,251.228,-87.704,173.832,29.955,155.422
C09719=1069.129,251.476,-87.732,173.834,29.959,155.423
C09720=1069.135,251.724,-87.760,173.836,29.963,155.424
C09721=1069.141,251.972,-87.788,173.839,29.967,155.425
C09722=1069.147,252.221,-87.816,173.841,29.971,155.425
C09723=1069.152,252.469,-87.844,173.844,29.975,155.426
C09724=1069.158,252.718,-87.872,173.846,29.979,155.427
C09725=1069.165,252.966,-87.900,173.848,29.983,155.427
C09726=1069.170,253.214,-87.928,173.851,29.987,155.428
C09727=1069.176,253.463,-87.956,173.853,29.991,155.429
C09728=1069.182,253.711,-87.984,173.856,29.995,155.429
C09729=1069.188,253.959,-88.012,173.859,29.999,155.430
C09730=1069.194,254.208,-88.040,173.860,30.003,155.431
C09731=1069.200,254.456,-88.068,173.863,30.007,155.431
C09732=1069.206,254.704,-88.097,173.865,30.011,155.432
C09733=1069.212,254.953,-88.126,173.868,30.015,155.433
C09734=1069.218,255.201,-88.153,173.871,30.019,155.433
C09735=1069.224,255.450,-88.181,173.873,30.023,155.434
C09736=1069.230,255.698,-88.210,173.875,30.027,155.435
C09737=1069.235,255.946,-88.238,173.877,30.031,155.435
C09738=1069.241,256.195,-88.267,173.880,30.035,155.436
C09739=1069.248,256.443,-88.294,173.883,30.039,155.437
C09740=1069.254,256.692,-88.323,173.885,30.043,155.437
C09741=1069.259,256.940,-88.351,173.888,30.046,155.438
C09742=1069.266,257.188,-88.380,173.890,30.051,155.439
C09743=1069.271,257.437,-88.408,173.892,30.055,155.439
C09744=1069.277,257.685,-88.436,173.895,30.058,155.440
C09745=1069.284,257.933,-88.464,173.897,30.062,155.441
C09746=1069.290,258.181,-88.493,173.900,30.066,155.441
C09747=1069.296,258.430,-88.521,173.902,30.070,155.442
C09748=1069.301,258.678,-88.550,173.905,30.075,155.443
C09749=1069.307,258.926,-88.578,173.908,30.079,155.443
C09750=1069.313,259.175,-88.606,173.910,30.082,155.444
C09751=1069.320,259.423,-88.635,173.912,30.086,155.445
C09752=1069.326,259.672,-88.663,173.914,30.090,155.445
C09753=1069.332,259.919,-88.692,173.917,30.094,155.446
C09754=1069.338,260.168,-88.720,173.920,30.098,155.447
C09755=1069.344,260.416,-88.749,173.922,30.102,155.447
C09756=1069.350,260.665,-88.778,173.925,30.106,155.448
C09757=1069.356,260.913,-88.806,173.927,30.110,155.449
C09758=1069.362,261.161,-88.834,173.930,30.114,155.449
C09759=1069.368,261.409,-88.862,173.933,30.118,155.450
C09760=1069.374,261.657,-88.891,173.935,30.122,155.451
C09761=1069.381,261.906,-88.920,173.937,30.125,155.451
C09762=1069.387,262.154,-88.949,173.940,30.129,155.452
C09763=1069.397,262.575,-88.997,173.944,30.136,155.453
C09764=1069.407,262.994,-89.046,173.948,30.143,155.454
C09765=1069.418,263.414,-89.094,173.953,30.149,155.455
C09766=1069.428,263.833,-89.143,173.957,30.156,155.457
C09767=1069.434,264.082,-89.171,173.959,30.160,155.457
C09768=1069.439,264.331,-89.201,173.962,30.164,155.458
C09769=1069.446,264.579,-89.230,173.965,30.168,155.459
C09770=1069.451,264.827,-89.258,173.967,30.172,155.459
C09771=1069.457,265.075,-89.287,173.970,30.176,155.460
C09772=1069.464,265.323,-89.316,173.973,30.180,155.461
C09773=1069.469,265.571,-89.345,173.975,30.184,155.461
C09774=1069.475,265.820,-89.374,173.977,30.188,155.462
C09775=1069.481,266.068,-89.403,173.979,30.192,155.463
C09776=1069.488,266.316,-89.432,173.982,30.196,155.463
C09777=1069.494,266.565,-89.461,173.985,30.200,155.464
C09778=1069.499,266.812,-89.490,173.987,30.204,155.465
C09779=1069.505,267.061,-89.518,173.990,30.208,155.466
C09780=1069.511,267.309,-89.547,173.992,30.212,155.466
C09781=1069.517,267.557,-89.577,173.995,30.216,155.467
C09782=1069.523,267.806,-89.606,173.998,30.220,155.468
C09783=1069.529,268.054,-89.635,174.000,30.224,155.468
C09784=1069.535,268.302,-89.664,174.003,30.228,155.469
C09785=1069.541,268.550,-89.693,174.006,30.232,155.470
C09786=1069.547,268.799,-89.723,174.008,30.236,155.470
C09787=1069.553,269.047,-89.752,174.011,30.240,155.471
C09788=1069.559,269.295,-89.781,174.013,30.244,155.472
C09789=1069.565,269.543,-89.811,174.016,30.248,155.472
C09790=1069.571,269.791,-89.840,174.019,30.252,155.473
C09791=1069.577,270.040,-89.869,174.021,30.256,155.474
C09792=1069.583,270.288,-89.898,174.024,30.260,155.474
C09793=1069.589,270.536,-89.927,174.027,30.264,155.475
C09794=1069.595,270.784,-89.956,174.029,30.268,155.476
C09795=1069.601,271.033,-89.986,174.032,30.272,155.477
C09796=1069.607,271.281,-90.015,174.034,30.277,155.477
C09797=1069.613,271.529,-90.045,174.037,30.280,155.478
C09798=1069.619,271.777,-90.074,174.039,30.284,155.479
C09799=1069.624,272.026,-90.103,174.041,30.288,155.479
C09800=1069.631,272.274,-90.132,174.044,30.292,155.480
C09801=1069.637,272.522,-90.162,174.047,30.296,155.481
C09802=1069.643,272.770,-90.192,174.049,30.300,155.481
C09803=1069.649,273.018,-90.221,174.052,30.304,155.482
C09804=1069.655,273.267,-90.251,174.054,30.308,155.483
C09805=1069.661,273.515,-90.280,174.057,30.312,155.483
C09806=1069.666,273.763,-90.309,174.060,30.317,155.484
C09807=1069.673,274.011,-90.339,174.062,30.320,155.485
C09808=1069.678,274.259,-90.369,174.065,30.324,155.486
C09809=1069.685,274.507,-90.398,174.068,30.329,155.486
C09810=1069.690,274.755,-90.428,174.070,30.333,155.487
C09811=1069.696,275.003,-90.458,174.073,30.336,155.488
C09812=1069.702,275.252,-90.487,174.075,30.341,155.488
C09813=1069.708,275.499,-90.517,174.078,30.345,155.489
C09814=1069.714,275.748,-90.546,174.082,30.349,155.490
C09815=1069.719,275.959,-90.571,174.083,30.352,155.490
C09816=1069.725,276.171,-90.597,174.086,30.356,155.491
C09817=1069.729,276.383,-90.622,174.088,30.359,155.492
C09818=1069.734,276.595,-90.647,174.090,30.363,155.492
C09819=1069.739,276.806,-90.673,174.092,30.366,155.493
C09820=1069.745,277.018,-90.698,174.095,30.370,155.493
C09821=1069.750,277.229,-90.723,174.098,30.373,155.494
C09822=1069.755,277.441,-90.749,174.099,30.377,155.495
C09823=1069.761,277.689,-90.779,174.102,30.380,155.495
C09824=1069.766,277.937,-90.809,174.104,30.385,155.496
C09825=1069.773,278.185,-90.838,174.107,30.389,155.497
C09826=1069.779,278.434,-90.868,174.110,30.393,155.497
C09827=1069.785,278.682,-90.899,174.112,30.397,155.498
C09828=1069.791,278.930,-90.928,174.115,30.401,155.499
C09829=1069.797,279.178,-90.958,174.118,30.405,155.499
C09830=1069.802,279.426,-90.988,174.120,30.409,155.500
C09831=1069.809,279.673,-91.018,174.124,30.413,155.501
C09832=1069.815,279.923,-91.048,174.127,30.417,155.502
C09833=1069.821,280.170,-91.078,174.129,30.421,155.502
C09834=1069.828,280.418,-91.108,174.132,30.425,155.503
C09835=1069.833,280.666,-91.137,174.134,30.430,155.504
C09836=1069.839,280.914,-91.168,174.137,30.433,155.504
C09837=1069.845,281.162,-91.198,174.140,30.438,155.505
C09838=1069.851,281.411,-91.228,174.142,30.442,155.506
C09839=1069.857,281.659,-91.258,174.145,30.446,155.507
C09840=1069.862,281.907,-91.289,174.148,30.450,155.507
C09841=1069.868,282.155,-91.318,174.150,30.454,155.508
C09842=1069.874,282.403,-91.348,174.153,30.458,155.509
C09843=1069.881,282.651,-91.379,174.156,30.462,155.509
C09844=1069.887,282.899,-91.409,174.158,30.466,155.510
C09845=1069.892,283.148,-91.439,174.161,30.470,155.511
C09846=1069.898,283.395,-91.469,174.164,30.475,155.512
C09847=1069.904,283.643,-91.500,174.167,30.479,155.512
C09848=1069.910,283.892,-91.530,174.170,30.483,155.513
C09849=1069.916,284.140,-91.561,174.172,30.487,155.514
C09850=1069.922,284.387,-91.591,174.175,30.491,155.514
C09851=1069.928,284.636,-91.622,174.178,30.495,155.515
C09852=1069.935,284.884,-91.651,174.180,30.499,155.516
C09853=1069.940,285.132,-91.681,174.183,30.503,155.517
C09854=1069.946,285.380,-91.711,174.186,30.508,155.517
C09855=1069.953,285.628,-91.742,174.188,30.511,155.518
C09856=1069.958,285.876,-91.772,174.192,30.516,155.519
C09857=1069.964,286.124,-91.803,174.195,30.520,155.519
C09858=1069.971,286.372,-91.834,174.197,30.524,155.520
C09859=1069.977,286.620,-91.864,174.200,30.528,155.521
C09860=1069.982,286.868,-91.894,174.203,30.532,155.522
C09861=1069.989,287.117,-91.925,174.205,30.536,155.522
C09862=1069.995,287.364,-91.955,174.208,30.541,155.523
C09863=1070.000,287.612,-91.986,174.211,30.544,155.524
C09864=1070.007,287.861,-92.016,174.214,30.549,155.524
C09865=1070.013,288.109,-92.047,174.217,30.553,155.525
C09866=1070.018,288.356,-92.077,174.219,30.557,155.526
C09867=1070.025,288.604,-92.108,174.222,30.561,155.527
C09868=1070.031,288.852,-92.139,174.225,30.565,155.527
C09869=1070.037,289.101,-92.170,174.227,30.569,155.528
C09870=1070.043,289.348,-92.200,174.230,30.574,155.529
C09871=1070.048,289.565,-92.227,174.233,30.577,155.529
C09872=1070.054,289.781,-92.254,174.235,30.581,155.530
C09873=1070.059,289.999,-92.280,174.238,30.584,155.531
C09874=1070.064,290.216,-92.307,174.240,30.588,155.531
C09875=1070.069,290.432,-92.334,174.243,30.591,155.532
C09876=1070.075,290.649,-92.361,174.245,30.595,155.533
C09877=1070.080,290.866,-92.388,174.248,30.599,155.533
C09878=1070.085,291.082,-92.415,174.250,30.603,155.534
C09879=1070.091,291.331,-92.446,174.253,30.607,155.535
C09880=1070.097,291.579,-92.477,174.256,30.611,155.535
C09881=1070.103,291.827,-92.507,174.259,30.615,155.536
C09882=1070.109,292.074,-92.538,174.261,30.619,155.537
C09883=1070.115,292.323,-92.569,174.264,30.624,155.538
C09884=1070.121,292.571,-92.600,174.267,30.627,155.538
C09885=1070.127,292.818,-92.631,174.270,30.632,155.539
C09886=1070.134,293.067,-92.662,174.273,30.636,155.540
C09887=1070.139,293.314,-92.693,174.276,30.640,155.540
C09888=1070.145,293.563,-92.724,174.278,30.644,155.541
C09889=1070.151,293.810,-92.755,174.281,30.649,155.542
C09890=1070.158,294.059,-92.786,174.284,30.653,155.543
C09891=1070.163,294.307,-92.817,174.287,30.657,155.543
C09892=1070.170,294.555,-92.848,174.290,30.661,155.544
C09893=1070.176,294.802,-92.879,174.292,30.665,155.545
C09894=1070.182,295.050,-92.910,174.295,30.670,155.546
C09895=1070.187,295.298,-92.941,174.298,30.673,155.546
C09896=1070.194,295.546,-92.972,174.301,30.678,155.547
C09897=1070.200,295.794,-93.004,174.304,30.682,155.548
C09898=1070.206,296.042,-93.035,174.307,30.687,155.549
C09899=1070.212,296.290,-93.066,174.309,30.691,155.549
C09900=1070.218,296.538,-93.097,174.313,30.695,155.550
C09901=1070.224,296.786,-93.128,174.316,30.699,155.551
C09902=1070.230,297.033,-93.160,174.318,30.703,155.552
C09903=1070.236,297.282,-93.191,174.321,30.708,155.552
C09904=1070.242,297.530,-93.222,174.324,30.712,155.553
C09905=1070.248,297.777,-93.254,174.327,30.716,155.554
C09906=1070.253,298.026,-93.285,174.330,30.721,155.555
C09907=1070.259,298.273,-93.316,174.333,30.725,155.556
C09908=1070.265,298.521,-93.348,174.335,30.729,155.556
C09909=1070.272,298.768,-93.379,174.338,30.733,155.557
C09910=1070.278,299.017,-93.411,174.342,30.738,155.558
C09911=1070.283,299.265,-93.442,174.344,30.742,155.559
C09912=1070.289,299.513,-93.474,174.347,30.746,155.559
C09913=1070.295,299.761,-93.506,174.350,30.751,155.560
C09914=1070.301,300.008,-93.537,174.353,30.755,155.561
C09915=1070.307,300.256,-93.569,174.356,30.760,155.562
C09916=1070.313,300.504,-93.600,174.359,30.764,155.562
C09917=1070.319,300.752,-93.632,174.361,30.768,155.563
C09918=1070.324,301.000,-93.663,174.365,30.772,155.564
C09919=1070.331,301.248,-93.695,174.368,30.777,155.565
C09920=1070.337,301.496,-93.727,174.370,30.781,155.565
C09921=1070.342,301.744,-93.759,174.373,30.785,155.566
C09922=1070.349,301.992,-93.790,174.377,30.790,155.567
C09923=1070.354,302.239,-93.822,174.379,30.794,155.568
C09924=1070.360,302.487,-93.854,174.382,30.799,155.569
C09925=1070.367,302.735,-93.885,174.385,30.803,155.569
C09926=1070.372,302.983,-93.917,174.388,30.807,155.570
C09927=1070.378,303.207,-93.946,174.391,30.811,155.571
C09928=1070.383,303.431,-93.975,174.394,30.815,155.571
C09929=1070.388,303.655,-94.003,174.396,30.819,155.572
C09930=1070.394,303.880,-94.033,174.399,30.823,155.573
C09931=1070.400,304.104,-94.060,174.402,30.827,155.574
C09932=1070.405,304.327,-94.089,174.405,30.831,155.574
C09933=1070.411,304.552,-94.119,174.407,30.835,155.575
C09934=1070.416,304.776,-94.147,174.410,30.839,155.576
C09935=1070.422,305.024,-94.179,174.413,30.843,155.577
C09936=1070.428,305.272,-94.212,174.415,30.847,155.577
C09937=1070.434,305.519,-94.243,174.418,30.852,155.578
C09938=1070.440,305.767,-94.275,174.422,30.856,155.579
C09939=1070.446,306.016,-94.307,174.424,30.861,155.580
C09940=1070.452,306.264,-94.339,174.427,30.865,155.580
C09941=1070.459,306.510,-94.371,174.431,30.869,155.581
C09942=1070.465,306.759,-94.403,174.433,30.874,155.582
C09943=1070.471,307.007,-94.435,174.436,30.878,155.583
C09944=1070.477,307.254,-94.468,174.440,30.883,155.584
C09945=1070.483,307.503,-94.500,174.442,30.887,155.584
C09946=1070.489,307.750,-94.531,174.445,30.891,155.585
C09947=1070.495,307.997,-94.563,174.449,30.896,155.586
C09948=1070.501,308.246,-94.595,174.451,30.900,155.587
C09949=1070.507,308.494,-94.628,174.454,30.904,155.588
C09950=1070.514,308.741,-94.660,174.458,30.909,155.588
C09951=1070.520,308.989,-94.692,174.461,30.913,155.589
C09952=1070.527,309.237,-94.724,174.463,30.917,155.590
C09953=1070.532,309.484,-94.756,174.467,30.922,155.591
C09954=1070.538,309.733,-94.788,174.470,30.926,155.591
C09955=1070.544,309.980,-94.821,174.473,30.931,155.592
C09956=1070.550,310.228,-94.853,174.476,30.935,155.593
C09957=1070.557,310.476,-94.885,174.479,30.939,155.594
C09958=1070.563,310.724,-94.917,174.482,30.944,155.595
C09959=1070.570,310.972,-94.950,174.485,30.948,155.595
C09960=1070.576,311.220,-94.982,174.488,30.952,155.596
C09961=1070.582,311.467,-95.015,174.491,30.957,155.597
C09962=1070.588,311.715,-95.047,174.494,30.961,155.598
C09963=1070.594,311.963,-95.079,174.497,30.966,155.599
C09964=1070.600,312.211,-95.112,174.500,30.970,155.599
C09965=1070.607,312.459,-95.144,174.503,30.974,155.600
C09966=1070.613,312.706,-95.176,174.507,30.979,155.601
C09967=1070.620,312.954,-95.209,174.510,30.983,155.602
C09968=1070.626,313.202,-95.241,174.512,30.987,155.602
C09969=1070.632,313.450,-95.274,174.516,30.992,155.603
C09970=1070.638,313.697,-95.307,174.519,30.997,155.604
C09971=1070.644,313.945,-95.339,174.522,31.001,155.605
C09972=1070.651,314.193,-95.371,174.525,31.006,155.606
C09973=1070.657,314.441,-95.404,174.528,31.010,155.607
C09974=1070.663,314.688,-95.437,174.531,31.014,155.607
C09975=1070.668,314.937,-95.469,174.534,31.019,155.608
C09976=1070.675,315.184,-95.502,174.538,31.024,155.609
C09977=1070.681,315.432,-95.535,174.540,31.028,155.610
C09978=1070.687,315.680,-95.568,174.543,31.033,155.611
C09979=1070.693,315.927,-95.601,174.547,31.037,155.611
C09980=1070.699,316.175,-95.634,174.549,31.042,155.612
C09981=1070.705,316.423,-95.667,174.553,31.047,155.613
C09982=1070.711,316.671,-95.700,174.556,31.051,155.614
C09983=1070.716,316.897,-95.729,174.559,31.056,155.615
C09984=1070.722,317.123,-95.759,174.561,31.059,155.616
C09985=1070.727,317.348,-95.790,174.564,31.064,155.616
C09986=1070.732,317.574,-95.820,174.567,31.068,155.617
C09987=1070.738,317.800,-95.850,174.570,31.072,155.618
C09988=1070.743,318.026,-95.880,174.573,31.077,155.619
C09989=1070.749,318.251,-95.910,174.576,31.081,155.619
C09990=1070.754,318.477,-95.939,174.579,31.085,155.620
C09991=1070.760,318.725,-95.973,174.581,31.090,155.621
C09992=1070.766,318.973,-96.006,174.585,31.094,155.622
C09993=1070.773,319.221,-96.040,174.588,31.099,155.623
C09994=1070.779,319.469,-96.073,174.591,31.103,155.624
C09995=1070.785,319.716,-96.106,174.594,31.108,155.625
C09996=1070.791,319.964,-96.139,174.597,31.112,155.625
//INST
///DATE 2021/06/17 10:55
///ATTR SC,RW,RJ
////FRAME ROBOT
///GROUP1 RB1
NOP
MOVL C00000 V=800.0 PL=0
MOVL C00001 V=800.0 PL=0
MOVL C00002 V=800.0 PL=0
MOVL C00003 V=800.0 PL=0
MOVL C00004 V=800.0 PL=0
MOVL C00005 V=800.0 PL=0
MOVL C00006 V=800.0 PL=0
MOVL C00007 V=800.0 PL=0
MOVL C00008 V=800.0 PL=0
MOVL C00009 V=800.0 PL=0
MOVL C00010 V=800.0 PL=0
MOVL C00011 V=800.0 PL=0
MOVL C00012 V=800.0 PL=0
MOVL C00013 V=800.0 PL=0
MOVL C00014 V=800.0 PL=0
MOVL C00015 V=800.0 PL=0
MOVL C00016 V=800.0 PL=0
MOVL C00017 V=800.0 PL=0
MOVL C00018 V=800.0 PL=0
MOVL C00019 V=800.0 PL=0
MOVL C00020 V=800.0 PL=0
MOVL C00021 V=800.0 PL=0
MOVL C00022 V=800.0 PL=0
MOVL C00023 V=800.0 PL=0
MOVL C00024 V=800.0 PL=0
MOVL C00025 V=800.0 PL=0
MOVL C00026 V=800.0 PL=0
MOVL C00027 V=800.0 PL=0
MOVL C00028 V=800.0 PL=0
MOVL C00029 V=800.0 PL=0
MOVL C00030 V=800.0 PL=0
MOVL C00031 V=800.0 PL=0
MOVL C00032 V=800.0 PL=0
MOVL C00033 V=800.0 PL=0
MOVL C00034 V=800.0 PL=0
MOVL C00035 V=800.0 PL=0
MOVL C00036 V=800.0 PL=0
MOVL C00037 V=800.0 PL=0
MOVL C00038 V=800.0 PL=0
MOVL C00039 V=800.0 PL=0
MOVL C00040 V=800.0 PL=0
MOVL C00041 V=800.0 PL=0
MOVL C00042 V=800.0 PL=0
MOVL C00043 V=800.0 PL=0
MOVL C00044 V=800.0 PL=0
MOVL C00045 V=800.0 PL=0
MOVL C00046 V=800.0 PL=0
MOVL C00047 V=800.0 PL=0
MOVL C00048 V=800.0 PL=0
MOVL C00049 V=800.0 PL=0
MOVL C00050 V=800.0 PL=0
MOVL C00051 V=800.0 PL=0
MOVL C00052 V=800.0 PL=0
MOVL C00053 V=800.0 PL=0
MOVL C00054 V=800.0 PL=0
MOVL C00055 V=800.0 PL=0
MOVL C00056 V=800.0 PL=0
MOVL C00057 V=800.0 PL=0
MOVL C00058 V=800.0 PL=0
MOVL C00059 V=800.0 PL=0
MOVL C00060 V=800.0 PL=0
MOVL C00061 V=800.0 PL=0
MOVL C00062 V=800.0 PL=0
MOVL C00063 V=800.0 PL=0
MOVL C00064 V=800.0 PL=0
MOVL C00065 V=800.0 PL=0
MOVL C00066 V=800.0 PL=0
MOVL C00067 V=800.0 PL=0
MOVL C00068 V=800.0 PL=0
MOVL C00069 V=800.0 PL=0
MOVL C00070 V=800.0 PL=0
MOVL C00071 V=800.0 PL=0
MOVL C00072 V=800.0 PL=0
MOVL C00073 V=800.0 PL=0
MOVL C00074 V=800.0 PL=0
MOVL C00075 V=800.0 PL=0
MOVL C00076 V=800.0 PL=0
MOVL C00077 V=800.0 PL=0
MOVL C00078 V=800.0 PL=0
MOVL C00079 V=800.0 PL=0
MOVL C00080 V=800.0 PL=0
MOVL C00081 V=800.0 PL=0
MOVL C00082 V=800.0 PL=0
MOVL C00083 V=800.0 PL=0
MOVL C00084 V=800.0 PL=0
MOVL C00085 V=800.0 PL=0
MOVL C00086 V=800.0 PL=0
MOVL C00087 V=800.0 PL=0
MOVL C00088 V=800.0 PL=0
MOVL C00089 V=800.0 PL=0
MOVL C00090 V=800.0 PL=0
MOVL C00091 V=800.0 PL=0
MOVL C00092 V=800.0 PL=0
MOVL C00093 V=800.0 PL=0
MOVL C00094 V=800.0 PL=0
MOVL C00095 V=800.0 PL=0
MOVL C00096 V=800.0 PL=0
MOVL C00097 V=800.0 PL=0
MOVL C00098 V=800.0 PL=0
MOVL C00099 V=800.0 PL=0
MOVL C00100 V=800.0 PL=0
MOVL C00101 V=800.0 PL=0
MOVL C00102 V=800.0 PL=0
MOVL C00103 V=800.0 PL=0
MOVL C00104 V=800.0 PL=0
MOVL C00105 V=800.0 PL=0
MOVL C00106 V=800.0 PL=0
MOVL C00107 V=800.0 PL=0
MOVL C00108 V=800.0 PL=0
MOVL C00109 V=800.0 PL=0
MOVL C00110 V=800.0 PL=0
MOVL C00111 V=800.0 PL=0
MOVL C00112 V=800.0 PL=0
MOVL C00113 V=800.0 PL=0
MOVL C00114 V=800.0 PL=0
MOVL C00115 V=800.0 PL=0
MOVL C00116 V=800.0 PL=0
MOVL C00117 V=800.0 PL=0
MOVL C00118 V=800.0 PL=0
MOVL C00119 V=800.0 PL=0
MOVL C00120 V=800.0 PL=0
MOVL C00121 V=800.0 PL=0
MOVL C00122 V=800.0 PL=0
MOVL C00123 V=800.0 PL=0
MOVL C00124 V=800.0 PL=0
MOVL C00125 V=800.0 PL=0
MOVL C00126 V=800.0 PL=0
MOVL C00127 V=800.0 PL=0
MOVL C00128 V=800.0 PL=0
MOVL C00129 V=800.0 PL=0
MOVL C00130 V=800.0 PL=0
MOVL C00131 V=800.0 PL=0
MOVL C00132 V=800.0 PL=0
MOVL C00133 V=800.0 PL=0
MOVL C00134 V=800.0 PL=0
MOVL C00135 V=800.0 PL=0
MOVL C00136 V=800.0 PL=0
MOVL C00137 V=800.0 PL=0
MOVL C00138 V=800.0 PL=0
MOVL C00139 V=800.0 PL=0
MOVL C00140 V=800.0 PL=0
MOVL C00141 V=800.0 PL=0
MOVL C00142 V=800.0 PL=0
MOVL C00143 V=800.0 PL=0
MOVL C00144 V=800.0 PL=0
MOVL C00145 V=800.0 PL=0
MOVL C00146 V=800.0 PL=0
MOVL C00147 V=800.0 PL=0
MOVL C00148 V=800.0 PL=0
MOVL C00149 V=800.0 PL=0
MOVL C00150 V=800.0 PL=0
MOVL C00151 V=800.0 PL=0
MOVL C00152 V=800.0 PL=0
MOVL C00153 V=800.0 PL=0
MOVL C00154 V=800.0 PL=0
MOVL C00155 V=800.0 PL=0
MOVL C00156 V=800.0 PL=0
MOVL C00157 V=800.0 PL=0
MOVL C00158 V=800.0 PL=0
MOVL C00159 V=800.0 PL=0
MOVL C00160 V=800.0 PL=0
MOVL C00161 V=800.0 PL=0
MOVL C00162 V=800.0 PL=0
MOVL C00163 V=800.0 PL=0
MOVL C00164 V=800.0 PL=0
MOVL C00165 V=800.0 PL=0
MOVL C00166 V=800.0 PL=0
MOVL C00167 V=800.0 PL=0
MOVL C00168 V=800.0 PL=0
MOVL C00169 V=800.0 PL=0
MOVL C00170 V=800.0 PL=0
MOVL C00171 V=800.0 PL=0
MOVL C00172 V=800.0 PL=0
MOVL C00173 V=800.0 PL=0
MOVL C00174 V=800.0 PL=0
MOVL C00175 V=800.0 PL=0
MOVL C00176 V=800.0 PL=0
MOVL C00177 V=800.0 PL=0
MOVL C00178 V=800.0 PL=0
MOVL C00179 V=800.0 PL=0
MOVL C00180 V=800.0 PL=0
MOVL C00181 V=800.0 PL=0
MOVL C00182 V=800.0 PL=0
MOVL C00183 V=800.0 PL=0
MOVL C00184 V=800.0 PL=0
MOVL C00185 V=800.0 PL=0
MOVL C00186 V=800.0 PL=0
MOVL C00187 V=800.0 PL=0
MOVL C00188 V=800.0 PL=0
MOVL C00189 V=800.0 PL=0
MOVL C00190 V=800.0 PL=0
MOVL C00191 V=800.0 PL=0
MOVL C00192 V=800.0 PL=0
MOVL C00193 V=800.0 PL=0
MOVL C00194 V=800.0 PL=0
MOVL C00195 V=800.0 PL=0
MOVL C00196 V=800.0 PL=0
MOVL C00197 V=800.0 PL=0
MOVL C00198 V=800.0 PL=0
MOVL C00199 V=800.0 PL=0
MOVL C00200 V=800.0 PL=0
MOVL C00201 V=800.0 PL=0
MOVL C00202 V=800.0 PL=0
MOVL C00203 V=800.0 PL=0
MOVL C00204 V=800.0 PL=0
MOVL C00205 V=800.0 PL=0
MOVL C00206 V=800.0 PL=0
MOVL C00207 V=800.0 PL=0
MOVL C00208 V=800.0 PL=0
MOVL C00209 V=800.0 PL=0
MOVL C00210 V=800.0 PL=0
MOVL C00211 V=800.0 PL=0
MOVL C00212 V=800.0 PL=0
MOVL C00213 V=800.0 PL=0
MOVL C00214 V=800.0 PL=0
MOVL C00215 V=800.0 PL=0
MOVL C00216 V=800.0 PL=0
MOVL C00217 V=800.0 PL=0
MOVL C00218 V=800.0 PL=0
MOVL C00219 V=800.0 PL=0
MOVL C00220 V=800.0 PL=0
MOVL C00221 V=800.0 PL=0
MOVL C00222 V=800.0 PL=0
MOVL C00223 V=800.0 PL=0
MOVL C00224 V=800.0 PL=0
MOVL C00225 V=800.0 PL=0
MOVL C00226 V=800.0 PL=0
MOVL C00227 V=800.0 PL=0
MOVL C00228 V=800.0 PL=0
MOVL C00229 V=800.0 PL=0
MOVL C00230 V=800.0 PL=0
MOVL C00231 V=800.0 PL=0
MOVL C00232 V=800.0 PL=0
MOVL C00233 V=800.0 PL=0
MOVL C00234 V=800.0 PL=0
MOVL C00235 V=800.0 PL=0
MOVL C00236 V=800.0 PL=0
MOVL C00237 V=800.0 PL=0
MOVL C00238 V=800.0 PL=0
MOVL C00239 V=800.0 PL=0
MOVL C00240 V=800.0 PL=0
MOVL C00241 V=800.0 PL=0
MOVL C00242 V=800.0 PL=0
MOVL C00243 V=800.0 PL=0
MOVL C00244 V=800.0 PL=0
MOVL C00245 V=800.0 PL=0
MOVL C00246 V=800.0 PL=0
MOVL C00247 V=800.0 PL=0
MOVL C00248 V=800.0 PL=0
MOVL C00249 V=800.0 PL=0
MOVL C00250 V=800.0 PL=0
MOVL C00251 V=800.0 PL=0
MOVL C00252 V=800.0 PL=0
MOVL C00253 V=800.0 PL=0
MOVL C00254 V=800.0 PL=0
MOVL C00255 V=800.0 PL=0
MOVL C00256 V=800.0 PL=0
MOVL C00257 V=800.0 PL=0
MOVL C00258 V=800.0 PL=0
MOVL C00259 V=800.0 PL=0
MOVL C00260 V=800.0 PL=0
MOVL C00261 V=800.0 PL=0
MOVL C00262 V=800.0 PL=0
MOVL C00263 V=800.0 PL=0
MOVL C00264 V=800.0 PL=0
MOVL C00265 V=800.0 PL=0
MOVL C00266 V=800.0 PL=0
MOVL C00267 V=800.0 PL=0
MOVL C00268 V=800.0 PL=0
MOVL C00269 V=800.0 PL=0
MOVL C00270 V=800.0 PL=0
MOVL C00271 V=800.0 PL=0
MOVL C00272 V=800.0 PL=0
MOVL C00273 V=800.0 PL=0
MOVL C00274 V=800.0 PL=0
MOVL C00275 V=800.0 PL=0
MOVL C00276 V=800.0 PL=0
MOVL C00277 V=800.0 PL=0
MOVL C00278 V=800.0 PL=0
MOVL C00279 V=800.0 PL=0
MOVL C00280 V=800.0 PL=0
MOVL C00281 V=800.0 PL=0
MOVL C00282 V=800.0 PL=0
MOVL C00283 V=800.0 PL=0
MOVL C00284 V=800.0 PL=0
MOVL C00285 V=800.0 PL=0
MOVL C00286 V=800.0 PL=0
MOVL C00287 V=800.0 PL=0
MOVL C00288 V=800.0 PL=0
MOVL C00289 V=800.0 PL=0
MOVL C00290 V=800.0 PL=0
MOVL C00291 V=800.0 PL=0
MOVL C00292 V=800.0 PL=0
MOVL C00293 V=800.0 PL=0
MOVL C00294 V=800.0 PL=0
MOVL C00295 V=800.0 PL=0
MOVL C00296 V=800.0 PL=0
MOVL C00297 V=800.0 PL=0
MOVL C00298 V=800.0 PL=0
MOVL C00299 V=800.0 PL=0
MOVL C00300 V=800.0 PL=0
MOVL C00301 V=800.0 PL=0
MOVL C00302 V=800.0 PL=0
MOVL C00303 V=800.0 PL=0
MOVL C00304 V=800.0 PL=0
MOVL C00305 V=800.0 PL=0
MOVL C00306 V=800.0 PL=0
MOVL C00307 V=800.0 PL=0
MOVL C00308 V=800.0 PL=0
MOVL C00309 V=800.0 PL=0
MOVL C00310 V=800.0 PL=0
MOVL C00311 V=800.0 PL=0
MOVL C00312 V=800.0 PL=0
MOVL C00313 V=800.0 PL=0
MOVL C00314 V=800.0 PL=0
MOVL C00315 V=800.0 PL=0
MOVL C00316 V=800.0 PL=0
MOVL C00317 V=800.0 PL=0
MOVL C00318 V=800.0 PL=0
MOVL C00319 V=800.0 PL=0
MOVL C00320 V=800.0 PL=0
MOVL C00321 V=800.0 PL=0
MOVL C00322 V=800.0 PL=0
MOVL C00323 V=800.0 PL=0
MOVL C00324 V=800.0 PL=0
MOVL C00325 V=800.0 PL=0
MOVL C00326 V=800.0 PL=0
MOVL C00327 V=800.0 PL=0
MOVL C00328 V=800.0 PL=0
MOVL C00329 V=800.0 PL=0
MOVL C00330 V=800.0 PL=0
MOVL C00331 V=800.0 PL=0
MOVL C00332 V=800.0 PL=0
MOVL C00333 V=800.0 PL=0
MOVL C00334 V=800.0 PL=0
MOVL C00335 V=800.0 PL=0
MOVL C00336 V=800.0 PL=0
MOVL C00337 V=800.0 PL=0
MOVL C00338 V=800.0 PL=0
MOVL C00339 V=800.0 PL=0
MOVL C00340 V=800.0 PL=0
MOVL C00341 V=800.0 PL=0
MOVL C00342 V=800.0 PL=0
MOVL C00343 V=800.0 PL=0
MOVL C00344 V=800.0 PL=0
MOVL C00345 V=800.0 PL=0
MOVL C00346 V=800.0 PL=0
MOVL C00347 V=800.0 PL=0
MOVL C00348 V=800.0 PL=0
MOVL C00349 V=800.0 PL=0
MOVL C00350 V=800.0 PL=0
MOVL C00351 V=800.0 PL=0
MOVL C00352 V=800.0 PL=0
MOVL C00353 V=800.0 PL=0
MOVL C00354 V=800.0 PL=0
MOVL C00355 V=800.0 PL=0
MOVL C00356 V=800.0 PL=0
MOVL C00357 V=800.0 PL=0
MOVL C00358 V=800.0 PL=0
MOVL C00359 V=800.0 PL=0
MOVL C00360 V=800.0 PL=0
MOVL C00361 V=800.0 PL=0
MOVL C00362 V=800.0 PL=0
MOVL C00363 V=800.0 PL=0
MOVL C00364 V=800.0 PL=0
MOVL C00365 V=800.0 PL=0
MOVL C00366 V=800.0 PL=0
MOVL C00367 V=800.0 PL=0
MOVL C00368 V=800.0 PL=0
MOVL C00369 V=800.0 PL=0
MOVL C00370 V=800.0 PL=0
MOVL C00371 V=800.0 PL=0
MOVL C00372 V=800.0 PL=0
MOVL C00373 V=800.0 PL=0
MOVL C00374 V=800.0 PL=0
MOVL C00375 V=800.0 PL=0
MOVL C00376 V=800.0 PL=0
MOVL C00377 V=800.0 PL=0
MOVL C00378 V=800.0 PL=0
MOVL C00379 V=800.0 PL=0
MOVL C00380 V=800.0 PL=0
MOVL C00381 V=800.0 PL=0
MOVL C00382 V=800.0 PL=0
MOVL C00383 V=800.0 PL=0
MOVL C00384 V=800.0 PL=0
MOVL C00385 V=800.0 PL=0
MOVL C00386 V=800.0 PL=0
MOVL C00387 V=800.0 PL=0
MOVL C00388 V=800.0 PL=0
MOVL C00389 V=800.0 PL=0
MOVL C00390 V=800.0 PL=0
MOVL C00391 V=800.0 PL=0
MOVL C00392 V=800.0 PL=0
MOVL C00393 V=800.0 PL=0
MOVL C00394 V=800.0 PL=0
MOVL C00395 V=800.0 PL=0
MOVL C00396 V=800.0 PL=0
MOVL C00397 V=800.0 PL=0
MOVL C00398 V=800.0 PL=0
MOVL C00399 V=800.0 PL=0
MOVL C00400 V=800.0 PL=0
MOVL C00401 V=800.0 PL=0
MOVL C00402 V=800.0 PL=0
MOVL C00403 V=800.0 PL=0
MOVL C00404 V=800.0 PL=0
MOVL C00405 V=800.0 PL=0
MOVL C00406 V=800.0 PL=0
MOVL C00407 V=800.0 PL=0
MOVL C00408 V=800.0 PL=0
MOVL C00409 V=800.0 PL=0
MOVL C00410 V=800.0 PL=0
MOVL C00411 V=800.0 PL=0
MOVL C00412 V=800.0 PL=0
MOVL C00413 V=800.0 PL=0
MOVL C00414 V=800.0 PL=0
MOVL C00415 V=800.0 PL=0
MOVL C00416 V=800.0 PL=0
MOVL C00417 V=800.0 PL=0
MOVL C00418 V=800.0 PL=0
MOVL C00419 V=800.0 PL=0
MOVL C00420 V=800.0 PL=0
MOVL C00421 V=800.0 PL=0
MOVL C00422 V=800.0 PL=0
MOVL C00423 V=800.0 PL=0
MOVL C00424 V=800.0 PL=0
MOVL C00425 V=800.0 PL=0
MOVL C00426 V=800.0 PL=0
MOVL C00427 V=800.0 PL=0
MOVL C00428 V=800.0 PL=0
MOVL C00429 V=800.0 PL=0
MOVL C00430 V=800.0 PL=0
MOVL C00431 V=800.0 PL=0
MOVL C00432 V=800.0 PL=0
MOVL C00433 V=800.0 PL=0
MOVL C00434 V=800.0 PL=0
MOVL C00435 V=800.0 PL=0
MOVL C00436 V=800.0 PL=0
MOVL C00437 V=800.0 PL=0
MOVL C00438 V=800.0 PL=0
MOVL C00439 V=800.0 PL=0
MOVL C00440 V=800.0 PL=0
MOVL C00441 V=800.0 PL=0
MOVL C00442 V=800.0 PL=0
MOVL C00443 V=800.0 PL=0
MOVL C00444 V=800.0 PL=0
MOVL C00445 V=800.0 PL=0
MOVL C00446 V=800.0 PL=0
MOVL C00447 V=800.0 PL=0
MOVL C00448 V=800.0 PL=0
MOVL C00449 V=800.0 PL=0
MOVL C00450 V=800.0 PL=0
MOVL C00451 V=800.0 PL=0
MOVL C00452 V=800.0 PL=0
MOVL C00453 V=800.0 PL=0
MOVL C00454 V=800.0 PL=0
MOVL C00455 V=800.0 PL=0
MOVL C00456 V=800.0 PL=0
MOVL C00457 V=800.0 PL=0
MOVL C00458 V=800.0 PL=0
MOVL C00459 V=800.0 PL=0
MOVL C00460 V=800.0 PL=0
MOVL C00461 V=800.0 PL=0
MOVL C00462 V=800.0 PL=0
MOVL C00463 V=800.0 PL=0
MOVL C00464 V=800.0 PL=0
MOVL C00465 V=800.0 PL=0
MOVL C00466 V=800.0 PL=0
MOVL C00467 V=800.0 PL=0
MOVL C00468 V=800.0 PL=0
MOVL C00469 V=800.0 PL=0
MOVL C00470 V=800.0 PL=0
MOVL C00471 V=800.0 PL=0
MOVL C00472 V=800.0 PL=0
MOVL C00473 V=800.0 PL=0
MOVL C00474 V=800.0 PL=0
MOVL C00475 V=800.0 PL=0
MOVL C00476 V=800.0 PL=0
MOVL C00477 V=800.0 PL=0
MOVL C00478 V=800.0 PL=0
MOVL C00479 V=800.0 PL=0
MOVL C00480 V=800.0 PL=0
MOVL C00481 V=800.0 PL=0
MOVL C00482 V=800.0 PL=0
MOVL C00483 V=800.0 PL=0
MOVL C00484 V=800.0 PL=0
MOVL C00485 V=800.0 PL=0
MOVL C00486 V=800.0 PL=0
MOVL C00487 V=800.0 PL=0
MOVL C00488 V=800.0 PL=0
MOVL C00489 V=800.0 PL=0
MOVL C00490 V=800.0 PL=0
MOVL C00491 V=800.0 PL=0
MOVL C00492 V=800.0 PL=0
MOVL C00493 V=800.0 PL=0
MOVL C00494 V=800.0 PL=0
MOVL C00495 V=800.0 PL=0
MOVL C00496 V=800.0 PL=0
MOVL C00497 V=800.0 PL=0
MOVL C00498 V=800.0 PL=0
MOVL C00499 V=800.0 PL=0
MOVL C00500 V=800.0 PL=0
MOVL C00501 V=800.0 PL=0
MOVL C00502 V=800.0 PL=0
MOVL C00503 V=800.0 PL=0
MOVL C00504 V=800.0 PL=0
MOVL C00505 V=800.0 PL=0
MOVL C00506 V=800.0 PL=0
MOVL C00507 V=800.0 PL=0
MOVL C00508 V=800.0 PL=0
MOVL C00509 V=800.0 PL=0
MOVL C00510 V=800.0 PL=0
MOVL C00511 V=800.0 PL=0
MOVL C00512 V=800.0 PL=0
MOVL C00513 V=800.0 PL=0
MOVL C00514 V=800.0 PL=0
MOVL C00515 V=800.0 PL=0
MOVL C00516 V=800.0 PL=0
MOVL C00517 V=800.0 PL=0
MOVL C00518 V=800.0 PL=0
MOVL C00519 V=800.0 PL=0
MOVL C00520 V=800.0 PL=0
MOVL C00521 V=800.0 PL=0
MOVL C00522 V=800.0 PL=0
MOVL C00523 V=800.0 PL=0
MOVL C00524 V=800.0 PL=0
MOVL C00525 V=800.0 PL=0
MOVL C00526 V=800.0 PL=0
MOVL C00527 V=800.0 PL=0
MOVL C00528 V=800.0 PL=0
MOVL C00529 V=800.0 PL=0
MOVL C00530 V=800.0 PL=0
MOVL C00531 V=800.0 PL=0
MOVL C00532 V=800.0 PL=0
MOVL C00533 V=800.0 PL=0
MOVL C00534 V=800.0 PL=0
MOVL C00535 V=800.0 PL=0
MOVL C00536 V=800.0 PL=0
MOVL C00537 V=800.0 PL=0
MOVL C00538 V=800.0 PL=0
MOVL C00539 V=800.0 PL=0
MOVL C00540 V=800.0 PL=0
MOVL C00541 V=800.0 PL=0
MOVL C00542 V=800.0 PL=0
MOVL C00543 V=800.0 PL=0
MOVL C00544 V=800.0 PL=0
MOVL C00545 V=800.0 PL=0
MOVL C00546 V=800.0 PL=0
MOVL C00547 V=800.0 PL=0
MOVL C00548 V=800.0 PL=0
MOVL C00549 V=800.0 PL=0
MOVL C00550 V=800.0 PL=0
MOVL C00551 V=800.0 PL=0
MOVL C00552 V=800.0 PL=0
MOVL C00553 V=800.0 PL=0
MOVL C00554 V=800.0 PL=0
MOVL C00555 V=800.0 PL=0
MOVL C00556 V=800.0 PL=0
MOVL C00557 V=800.0 PL=0
MOVL C00558 V=800.0 PL=0
MOVL C00559 V=800.0 PL=0
MOVL C00560 V=800.0 PL=0
MOVL C00561 V=800.0 PL=0
MOVL C00562 V=800.0 PL=0
MOVL C00563 V=800.0 PL=0
MOVL C00564 V=800.0 PL=0
MOVL C00565 V=800.0 PL=0
MOVL C00566 V=800.0 PL=0
MOVL C00567 V=800.0 PL=0
MOVL C00568 V=800.0 PL=0
MOVL C00569 V=800.0 PL=0
MOVL C00570 V=800.0 PL=0
MOVL C00571 V=800.0 PL=0
MOVL C00572 V=800.0 PL=0
MOVL C00573 V=800.0 PL=0
MOVL C00574 V=800.0 PL=0
MOVL C00575 V=800.0 PL=0
MOVL C00576 V=800.0 PL=0
MOVL C00577 V=800.0 PL=0
MOVL C00578 V=800.0 PL=0
MOVL C00579 V=800.0 PL=0
MOVL C00580 V=800.0 PL=0
MOVL C00581 V=800.0 PL=0
MOVL C00582 V=800.0 PL=0
MOVL C00583 V=800.0 PL=0
MOVL C00584 V=800.0 PL=0
MOVL C00585 V=800.0 PL=0
MOVL C00586 V=800.0 PL=0
MOVL C00587 V=800.0 PL=0
MOVL C00588 V=800.0 PL=0
MOVL C00589 V=800.0 PL=0
MOVL C00590 V=800.0 PL=0
MOVL C00591 V=800.0 PL=0
MOVL C00592 V=800.0 PL=0
MOVL C00593 V=800.0 PL=0
MOVL C00594 V=800.0 PL=0
MOVL C00595 V=800.0 PL=0
MOVL C00596 V=800.0 PL=0
MOVL C00597 V=800.0 PL=0
MOVL C00598 V=800.0 PL=0
MOVL C00599 V=800.0 PL=0
MOVL C00600 V=800.0 PL=0
MOVL C00601 V=800.0 PL=0
MOVL C00602 V=800.0 PL=0
MOVL C00603 V=800.0 PL=0
MOVL C00604 V=800.0 PL=0
MOVL C00605 V=800.0 PL=0
MOVL C00606 V=800.0 PL=0
MOVL C00607 V=800.0 PL=0
MOVL C00608 V=800.0 PL=0
MOVL C00609 V=800.0 PL=0
MOVL C00610 V=800.0 PL=0
MOVL C00611 V=800.0 PL=0
MOVL C00612 V=800.0 PL=0
MOVL C00613 V=800.0 PL=0
MOVL C00614 V=800.0 PL=0
MOVL C00615 V=800.0 PL=0
MOVL C00616 V=800.0 PL=0
MOVL C00617 V=800.0 PL=0
MOVL C00618 V=800.0 PL=0
MOVL C00619 V=800.0 PL=0
MOVL C00620 V=800.0 PL=0
MOVL C00621 V=800.0 PL=0
MOVL C00622 V=800.0 PL=0
MOVL C00623 V=800.0 PL=0
MOVL C00624 V=800.0 PL=0
MOVL C00625 V=800.0 PL=0
MOVL C00626 V=800.0 PL=0
MOVL C00627 V=800.0 PL=0
MOVL C00628 V=800.0 PL=0
MOVL C00629 V=800.0 PL=0
MOVL C00630 V=800.0 PL=0
MOVL C00631 V=800.0 PL=0
MOVL C00632 V=800.0 PL=0
MOVL C00633 V=800.0 PL=0
MOVL C00634 V=800.0 PL=0
MOVL C00635 V=800.0 PL=0
MOVL C00636 V=800.0 PL=0
MOVL C00637 V=800.0 PL=0
MOVL C00638 V=800.0 PL=0
MOVL C00639 V=800.0 PL=0
MOVL C00640 V=800.0 PL=0
MOVL C00641 V=800.0 PL=0
MOVL C00642 V=800.0 PL=0
MOVL C00643 V=800.0 PL=0
MOVL C00644 V=800.0 PL=0
MOVL C00645 V=800.0 PL=0
MOVL C00646 V=800.0 PL=0
MOVL C00647 V=800.0 PL=0
MOVL C00648 V=800.0 PL=0
MOVL C00649 V=800.0 PL=0
MOVL C00650 V=800.0 PL=0
MOVL C00651 V=800.0 PL=0
MOVL C00652 V=800.0 PL=0
MOVL C00653 V=800.0 PL=0
MOVL C00654 V=800.0 PL=0
MOVL C00655 V=800.0 PL=0
MOVL C00656 V=800.0 PL=0
MOVL C00657 V=800.0 PL=0
MOVL C00658 V=800.0 PL=0
MOVL C00659 V=800.0 PL=0
MOVL C00660 V=800.0 PL=0
MOVL C00661 V=800.0 PL=0
MOVL C00662 V=800.0 PL=0
MOVL C00663 V=800.0 PL=0
MOVL C00664 V=800.0 PL=0
MOVL C00665 V=800.0 PL=0
MOVL C00666 V=800.0 PL=0
MOVL C00667 V=800.0 PL=0
MOVL C00668 V=800.0 PL=0
MOVL C00669 V=800.0 PL=0
MOVL C00670 V=800.0 PL=0
MOVL C00671 V=800.0 PL=0
MOVL C00672 V=800.0 PL=0
MOVL C00673 V=800.0 PL=0
MOVL C00674 V=800.0 PL=0
MOVL C00675 V=800.0 PL=0
MOVL C00676 V=800.0 PL=0
MOVL C00677 V=800.0 PL=0
MOVL C00678 V=800.0 PL=0
MOVL C00679 V=800.0 PL=0
MOVL C00680 V=800.0 PL=0
MOVL C00681 V=800.0 PL=0
MOVL C00682 V=800.0 PL=0
MOVL C00683 V=800.0 PL=0
MOVL C00684 V=800.0 PL=0
MOVL C00685 V=800.0 PL=0
MOVL C00686 V=800.0 PL=0
MOVL C00687 V=800.0 PL=0
MOVL C00688 V=800.0 PL=0
MOVL C00689 V=800.0 PL=0
MOVL C00690 V=800.0 PL=0
MOVL C00691 V=800.0 PL=0
MOVL C00692 V=800.0 PL=0
MOVL C00693 V=800.0 PL=0
MOVL C00694 V=800.0 PL=0
MOVL C00695 V=800.0 PL=0
MOVL C00696 V=800.0 PL=0
MOVL C00697 V=800.0 PL=0
MOVL C00698 V=800.0 PL=0
MOVL C00699 V=800.0 PL=0
MOVL C00700 V=800.0 PL=0
MOVL C00701 V=800.0 PL=0
MOVL C00702 V=800.0 PL=0
MOVL C00703 V=800.0 PL=0
MOVL C00704 V=800.0 PL=0
MOVL C00705 V=800.0 PL=0
MOVL C00706 V=800.0 PL=0
MOVL C00707 V=800.0 PL=0
MOVL C00708 V=800.0 PL=0
MOVL C00709 V=800.0 PL=0
MOVL C00710 V=800.0 PL=0
MOVL C00711 V=800.0 PL=0
MOVL C00712 V=800.0 PL=0
MOVL C00713 V=800.0 PL=0
MOVL C00714 V=800.0 PL=0
MOVL C00715 V=800.0 PL=0
MOVL C00716 V=800.0 PL=0
MOVL C00717 V=800.0 PL=0
MOVL C00718 V=800.0 PL=0
MOVL C00719 V=800.0 PL=0
MOVL C00720 V=800.0 PL=0
MOVL C00721 V=800.0 PL=0
MOVL C00722 V=800.0 PL=0
MOVL C00723 V=800.0 PL=0
MOVL C00724 V=800.0 PL=0
MOVL C00725 V=800.0 PL=0
MOVL C00726 V=800.0 PL=0
MOVL C00727 V=800.0 PL=0
MOVL C00728 V=800.0 PL=0
MOVL C00729 V=800.0 PL=0
MOVL C00730 V=800.0 PL=0
MOVL C00731 V=800.0 PL=0
MOVL C00732 V=800.0 PL=0
MOVL C00733 V=800.0 PL=0
MOVL C00734 V=800.0 PL=0
MOVL C00735 V=800.0 PL=0
MOVL C00736 V=800.0 PL=0
MOVL C00737 V=800.0 PL=0
MOVL C00738 V=800.0 PL=0
MOVL C00739 V=800.0 PL=0
MOVL C00740 V=800.0 PL=0
MOVL C00741 V=800.0 PL=0
MOVL C00742 V=800.0 PL=0
MOVL C00743 V=800.0 PL=0
MOVL C00744 V=800.0 PL=0
MOVL C00745 V=800.0 PL=0
MOVL C00746 V=800.0 PL=0
MOVL C00747 V=800.0 PL=0
MOVL C00748 V=800.0 PL=0
MOVL C00749 V=800.0 PL=0
MOVL C00750 V=800.0 PL=0
MOVL C00751 V=800.0 PL=0
MOVL C00752 V=800.0 PL=0
MOVL C00753 V=800.0 PL=0
MOVL C00754 V=800.0 PL=0
MOVL C00755 V=800.0 PL=0
MOVL C00756 V=800.0 PL=0
MOVL C00757 V=800.0 PL=0
MOVL C00758 V=800.0 PL=0
MOVL C00759 V=800.0 PL=0
MOVL C00760 V=800.0 PL=0
MOVL C00761 V=800.0 PL=0
MOVL C00762 V=800.0 PL=0
MOVL C00763 V=800.0 PL=0
MOVL C00764 V=800.0 PL=0
MOVL C00765 V=800.0 PL=0
MOVL C00766 V=800.0 PL=0
MOVL C00767 V=800.0 PL=0
MOVL C00768 V=800.0 PL=0
MOVL C00769 V=800.0 PL=0
MOVL C00770 V=800.0 PL=0
MOVL C00771 V=800.0 PL=0
MOVL C00772 V=800.0 PL=0
MOVL C00773 V=800.0 PL=0
MOVL C00774 V=800.0 PL=0
MOVL C00775 V=800.0 PL=0
MOVL C00776 V=800.0 PL=0
MOVL C00777 V=800.0 PL=0
MOVL C00778 V=800.0 PL=0
MOVL C00779 V=800.0 PL=0
MOVL C00780 V=800.0 PL=0
MOVL C00781 V=800.0 PL=0
MOVL C00782 V=800.0 PL=0
MOVL C00783 V=800.0 PL=0
MOVL C00784 V=800.0 PL=0
MOVL C00785 V=800.0 PL=0
MOVL C00786 V=800.0 PL=0
MOVL C00787 V=800.0 PL=0
MOVL C00788 V=800.0 PL=0
MOVL C00789 V=800.0 PL=0
MOVL C00790 V=800.0 PL=0
MOVL C00791 V=800.0 PL=0
MOVL C00792 V=800.0 PL=0
MOVL C00793 V=800.0 PL=0
MOVL C00794 V=800.0 PL=0
MOVL C00795 V=800.0 PL=0
MOVL C00796 V=800.0 PL=0
MOVL C00797 V=800.0 PL=0
MOVL C00798 V=800.0 PL=0
MOVL C00799 V=800.0 PL=0
MOVL C00800 V=800.0 PL=0
MOVL C00801 V=800.0 PL=0
MOVL C00802 V=800.0 PL=0
MOVL C00803 V=800.0 PL=0
MOVL C00804 V=800.0 PL=0
MOVL C00805 V=800.0 PL=0
MOVL C00806 V=800.0 PL=0
MOVL C00807 V=800.0 PL=0
MOVL C00808 V=800.0 PL=0
MOVL C00809 V=800.0 PL=0
MOVL C00810 V=800.0 PL=0
MOVL C00811 V=800.0 PL=0
MOVL C00812 V=800.0 PL=0
MOVL C00813 V=800.0 PL=0
MOVL C00814 V=800.0 PL=0
MOVL C00815 V=800.0 PL=0
MOVL C00816 V=800.0 PL=0
MOVL C00817 V=800.0 PL=0
MOVL C00818 V=800.0 PL=0
MOVL C00819 V=800.0 PL=0
MOVL C00820 V=800.0 PL=0
MOVL C00821 V=800.0 PL=0
MOVL C00822 V=800.0 PL=0
MOVL C00823 V=800.0 PL=0
MOVL C00824 V=800.0 PL=0
MOVL C00825 V=800.0 PL=0
MOVL C00826 V=800.0 PL=0
MOVL C00827 V=800.0 PL=0
MOVL C00828 V=800.0 PL=0
MOVL C00829 V=800.0 PL=0
MOVL C00830 V=800.0 PL=0
MOVL C00831 V=800.0 PL=0
MOVL C00832 V=800.0 PL=0
MOVL C00833 V=800.0 PL=0
MOVL C00834 V=800.0 PL=0
MOVL C00835 V=800.0 PL=0
MOVL C00836 V=800.0 PL=0
MOVL C00837 V=800.0 PL=0
MOVL C00838 V=800.0 PL=0
MOVL C00839 V=800.0 PL=0
MOVL C00840 V=800.0 PL=0
MOVL C00841 V=800.0 PL=0
MOVL C00842 V=800.0 PL=0
MOVL C00843 V=800.0 PL=0
MOVL C00844 V=800.0 PL=0
MOVL C00845 V=800.0 PL=0
MOVL C00846 V=800.0 PL=0
MOVL C00847 V=800.0 PL=0
MOVL C00848 V=800.0 PL=0
MOVL C00849 V=800.0 PL=0
MOVL C00850 V=800.0 PL=0
MOVL C00851 V=800.0 PL=0
MOVL C00852 V=800.0 PL=0
MOVL C00853 V=800.0 PL=0
MOVL C00854 V=800.0 PL=0
MOVL C00855 V=800.0 PL=0
MOVL C00856 V=800.0 PL=0
MOVL C00857 V=800.0 PL=0
MOVL C00858 V=800.0 PL=0
MOVL C00859 V=800.0 PL=0
MOVL C00860 V=800.0 PL=0
MOVL C00861 V=800.0 PL=0
MOVL C00862 V=800.0 PL=0
MOVL C00863 V=800.0 PL=0
MOVL C00864 V=800.0 PL=0
MOVL C00865 V=800.0 PL=0
MOVL C00866 V=800.0 PL=0
MOVL C00867 V=800.0 PL=0
MOVL C00868 V=800.0 PL=0
MOVL C00869 V=800.0 PL=0
MOVL C00870 V=800.0 PL=0
MOVL C00871 V=800.0 PL=0
MOVL C00872 V=800.0 PL=0
MOVL C00873 V=800.0 PL=0
MOVL C00874 V=800.0 PL=0
MOVL C00875 V=800.0 PL=0
MOVL C00876 V=800.0 PL=0
MOVL C00877 V=800.0 PL=0
MOVL C00878 V=800.0 PL=0
MOVL C00879 V=800.0 PL=0
MOVL C00880 V=800.0 PL=0
MOVL C00881 V=800.0 PL=0
MOVL C00882 V=800.0 PL=0
MOVL C00883 V=800.0 PL=0
MOVL C00884 V=800.0 PL=0
MOVL C00885 V=800.0 PL=0
MOVL C00886 V=800.0 PL=0
MOVL C00887 V=800.0 PL=0
MOVL C00888 V=800.0 PL=0
MOVL C00889 V=800.0 PL=0
MOVL C00890 V=800.0 PL=0
MOVL C00891 V=800.0 PL=0
MOVL C00892 V=800.0 PL=0
MOVL C00893 V=800.0 PL=0
MOVL C00894 V=800.0 PL=0
MOVL C00895 V=800.0 PL=0
MOVL C00896 V=800.0 PL=0
MOVL C00897 V=800.0 PL=0
MOVL C00898 V=800.0 PL=0
MOVL C00899 V=800.0 PL=0
MOVL C00900 V=800.0 PL=0
MOVL C00901 V=800.0 PL=0
MOVL C00902 V=800.0 PL=0
MOVL C00903 V=800.0 PL=0
MOVL C00904 V=800.0 PL=0
MOVL C00905 V=800.0 PL=0
MOVL C00906 V=800.0 PL=0
MOVL C00907 V=800.0 PL=0
MOVL C00908 V=800.0 PL=0
MOVL C00909 V=800.0 PL=0
MOVL C00910 V=800.0 PL=0
MOVL C00911 V=800.0 PL=0
MOVL C00912 V=800.0 PL=0
MOVL C00913 V=800.0 PL=0
MOVL C00914 V=800.0 PL=0
MOVL C00915 V=800.0 PL=0
MOVL C00916 V=800.0 PL=0
MOVL C00917 V=800.0 PL=0
MOVL C00918 V=800.0 PL=0
MOVL C00919 V=800.0 PL=0
MOVL C00920 V=800.0 PL=0
MOVL C00921 V=800.0 PL=0
MOVL C00922 V=800.0 PL=0
MOVL C00923 V=800.0 PL=0
MOVL C00924 V=800.0 PL=0
MOVL C00925 V=800.0 PL=0
MOVL C00926 V=800.0 PL=0
MOVL C00927 V=800.0 PL=0
MOVL C00928 V=800.0 PL=0
MOVL C00929 V=800.0 PL=0
MOVL C00930 V=800.0 PL=0
MOVL C00931 V=800.0 PL=0
MOVL C00932 V=800.0 PL=0
MOVL C00933 V=800.0 PL=0
MOVL C00934 V=800.0 PL=0
MOVL C00935 V=800.0 PL=0
MOVL C00936 V=800.0 PL=0
MOVL C00937 V=800.0 PL=0
MOVL C00938 V=800.0 PL=0
MOVL C00939 V=800.0 PL=0
MOVL C00940 V=800.0 PL=0
MOVL C00941 V=800.0 PL=0
MOVL C00942 V=800.0 PL=0
MOVL C00943 V=800.0 PL=0
MOVL C00944 V=800.0 PL=0
MOVL C00945 V=800.0 PL=0
MOVL C00946 V=800.0 PL=0
MOVL C00947 V=800.0 PL=0
MOVL C00948 V=800.0 PL=0
MOVL C00949 V=800.0 PL=0
MOVL C00950 V=800.0 PL=0
MOVL C00951 V=800.0 PL=0
MOVL C00952 V=800.0 PL=0
MOVL C00953 V=800.0 PL=0
MOVL C00954 V=800.0 PL=0
MOVL C00955 V=800.0 PL=0
MOVL C00956 V=800.0 PL=0
MOVL C00957 V=800.0 PL=0
MOVL C00958 V=800.0 PL=0
MOVL C00959 V=800.0 PL=0
MOVL C00960 V=800.0 PL=0
MOVL C00961 V=800.0 PL=0
MOVL C00962 V=800.0 PL=0
MOVL C00963 V=800.0 PL=0
MOVL C00964 V=800.0 PL=0
MOVL C00965 V=800.0 PL=0
MOVL C00966 V=800.0 PL=0
MOVL C00967 V=800.0 PL=0
MOVL C00968 V=800.0 PL=0
MOVL C00969 V=800.0 PL=0
MOVL C00970 V=800.0 PL=0
MOVL C00971 V=800.0 PL=0
MOVL C00972 V=800.0 PL=0
MOVL C00973 V=800.0 PL=0
MOVL C00974 V=800.0 PL=0
MOVL C00975 V=800.0 PL=0
MOVL C00976 V=800.0 PL=0
MOVL C00977 V=800.0 PL=0
MOVL C00978 V=800.0 PL=0
MOVL C00979 V=800.0 PL=0
MOVL C00980 V=800.0 PL=0
MOVL C00981 V=800.0 PL=0
MOVL C00982 V=800.0 PL=0
MOVL C00983 V=800.0 PL=0
MOVL C00984 V=800.0 PL=0
MOVL C00985 V=800.0 PL=0
MOVL C00986 V=800.0 PL=0
MOVL C00987 V=800.0 PL=0
MOVL C00988 V=800.0 PL=0
MOVL C00989 V=800.0 PL=0
MOVL C00990 V=800.0 PL=0
MOVL C00991 V=800.0 PL=0
MOVL C00992 V=800.0 PL=0
MOVL C00993 V=800.0 PL=0
MOVL C00994 V=800.0 PL=0
MOVL C00995 V=800.0 PL=0
MOVL C00996 V=800.0 PL=0
MOVL C00997 V=800.0 PL=0
MOVL C00998 V=800.0 PL=0
MOVL C00999 V=800.0 PL=0
MOVL C01000 V=800.0 PL=0
MOVL C01001 V=800.0 PL=0
MOVL C01002 V=800.0 PL=0
MOVL C01003 V=800.0 PL=0
MOVL C01004 V=800.0 PL=0
MOVL C01005 V=800.0 PL=0
MOVL C01006 V=800.0 PL=0
MOVL C01007 V=800.0 PL=0
MOVL C01008 V=800.0 PL=0
MOVL C01009 V=800.0 PL=0
MOVL C01010 V=800.0 PL=0
MOVL C01011 V=800.0 PL=0
MOVL C01012 V=800.0 PL=0
MOVL C01013 V=800.0 PL=0
MOVL C01014 V=800.0 PL=0
MOVL C01015 V=800.0 PL=0
MOVL C01016 V=800.0 PL=0
MOVL C01017 V=800.0 PL=0
MOVL C01018 V=800.0 PL=0
MOVL C01019 V=800.0 PL=0
MOVL C01020 V=800.0 PL=0
MOVL C01021 V=800.0 PL=0
MOVL C01022 V=800.0 PL=0
MOVL C01023 V=800.0 PL=0
MOVL C01024 V=800.0 PL=0
MOVL C01025 V=800.0 PL=0
MOVL C01026 V=800.0 PL=0
MOVL C01027 V=800.0 PL=0
MOVL C01028 V=800.0 PL=0
MOVL C01029 V=800.0 PL=0
MOVL C01030 V=800.0 PL=0
MOVL C01031 V=800.0 PL=0
MOVL C01032 V=800.0 PL=0
MOVL C01033 V=800.0 PL=0
MOVL C01034 V=800.0 PL=0
MOVL C01035 V=800.0 PL=0
MOVL C01036 V=800.0 PL=0
MOVL C01037 V=800.0 PL=0
MOVL C01038 V=800.0 PL=0
MOVL C01039 V=800.0 PL=0
MOVL C01040 V=800.0 PL=0
MOVL C01041 V=800.0 PL=0
MOVL C01042 V=800.0 PL=0
MOVL C01043 V=800.0 PL=0
MOVL C01044 V=800.0 PL=0
MOVL C01045 V=800.0 PL=0
MOVL C01046 V=800.0 PL=0
MOVL C01047 V=800.0 PL=0
MOVL C01048 V=800.0 PL=0
MOVL C01049 V=800.0 PL=0
MOVL C01050 V=800.0 PL=0
MOVL C01051 V=800.0 PL=0
MOVL C01052 V=800.0 PL=0
MOVL C01053 V=800.0 PL=0
MOVL C01054 V=800.0 PL=0
MOVL C01055 V=800.0 PL=0
MOVL C01056 V=800.0 PL=0
MOVL C01057 V=800.0 PL=0
MOVL C01058 V=800.0 PL=0
MOVL C01059 V=800.0 PL=0
MOVL C01060 V=800.0 PL=0
MOVL C01061 V=800.0 PL=0
MOVL C01062 V=800.0 PL=0
MOVL C01063 V=800.0 PL=0
MOVL C01064 V=800.0 PL=0
MOVL C01065 V=800.0 PL=0
MOVL C01066 V=800.0 PL=0
MOVL C01067 V=800.0 PL=0
MOVL C01068 V=800.0 PL=0
MOVL C01069 V=800.0 PL=0
MOVL C01070 V=800.0 PL=0
MOVL C01071 V=800.0 PL=0
MOVL C01072 V=800.0 PL=0
MOVL C01073 V=800.0 PL=0
MOVL C01074 V=800.0 PL=0
MOVL C01075 V=800.0 PL=0
MOVL C01076 V=800.0 PL=0
MOVL C01077 V=800.0 PL=0
MOVL C01078 V=800.0 PL=0
MOVL C01079 V=800.0 PL=0
MOVL C01080 V=800.0 PL=0
MOVL C01081 V=800.0 PL=0
MOVL C01082 V=800.0 PL=0
MOVL C01083 V=800.0 PL=0
MOVL C01084 V=800.0 PL=0
MOVL C01085 V=800.0 PL=0
MOVL C01086 V=800.0 PL=0
MOVL C01087 V=800.0 PL=0
MOVL C01088 V=800.0 PL=0
MOVL C01089 V=800.0 PL=0
MOVL C01090 V=800.0 PL=0
MOVL C01091 V=800.0 PL=0
MOVL C01092 V=800.0 PL=0
MOVL C01093 V=800.0 PL=0
MOVL C01094 V=800.0 PL=0
MOVL C01095 V=800.0 PL=0
MOVL C01096 V=800.0 PL=0
MOVL C01097 V=800.0 PL=0
MOVL C01098 V=800.0 PL=0
MOVL C01099 V=800.0 PL=0
MOVL C01100 V=800.0 PL=0
MOVL C01101 V=800.0 PL=0
MOVL C01102 V=800.0 PL=0
MOVL C01103 V=800.0 PL=0
MOVL C01104 V=800.0 PL=0
MOVL C01105 V=800.0 PL=0
MOVL C01106 V=800.0 PL=0
MOVL C01107 V=800.0 PL=0
MOVL C01108 V=800.0 PL=0
MOVL C01109 V=800.0 PL=0
MOVL C01110 V=800.0 PL=0
MOVL C01111 V=800.0 PL=0
MOVL C01112 V=800.0 PL=0
MOVL C01113 V=800.0 PL=0
MOVL C01114 V=800.0 PL=0
MOVL C01115 V=800.0 PL=0
MOVL C01116 V=800.0 PL=0
MOVL C01117 V=800.0 PL=0
MOVL C01118 V=800.0 PL=0
MOVL C01119 V=800.0 PL=0
MOVL C01120 V=800.0 PL=0
MOVL C01121 V=800.0 PL=0
MOVL C01122 V=800.0 PL=0
MOVL C01123 V=800.0 PL=0
MOVL C01124 V=800.0 PL=0
MOVL C01125 V=800.0 PL=0
MOVL C01126 V=800.0 PL=0
MOVL C01127 V=800.0 PL=0
MOVL C01128 V=800.0 PL=0
MOVL C01129 V=800.0 PL=0
MOVL C01130 V=800.0 PL=0
MOVL C01131 V=800.0 PL=0
MOVL C01132 V=800.0 PL=0
MOVL C01133 V=800.0 PL=0
MOVL C01134 V=800.0 PL=0
MOVL C01135 V=800.0 PL=0
MOVL C01136 V=800.0 PL=0
MOVL C01137 V=800.0 PL=0
MOVL C01138 V=800.0 PL=0
MOVL C01139 V=800.0 PL=0
MOVL C01140 V=800.0 PL=0
MOVL C01141 V=800.0 PL=0
MOVL C01142 V=800.0 PL=0
MOVL C01143 V=800.0 PL=0
MOVL C01144 V=800.0 PL=0
MOVL C01145 V=800.0 PL=0
MOVL C01146 V=800.0 PL=0
MOVL C01147 V=800.0 PL=0
MOVL C01148 V=800.0 PL=0
MOVL C01149 V=800.0 PL=0
MOVL C01150 V=800.0 PL=0
MOVL C01151 V=800.0 PL=0
MOVL C01152 V=800.0 PL=0
MOVL C01153 V=800.0 PL=0
MOVL C01154 V=800.0 PL=0
MOVL C01155 V=800.0 PL=0
MOVL C01156 V=800.0 PL=0
MOVL C01157 V=800.0 PL=0
MOVL C01158 V=800.0 PL=0
MOVL C01159 V=800.0 PL=0
MOVL C01160 V=800.0 PL=0
MOVL C01161 V=800.0 PL=0
MOVL C01162 V=800.0 PL=0
MOVL C01163 V=800.0 PL=0
MOVL C01164 V=800.0 PL=0
MOVL C01165 V=800.0 PL=0
MOVL C01166 V=800.0 PL=0
MOVL C01167 V=800.0 PL=0
MOVL C01168 V=800.0 PL=0
MOVL C01169 V=800.0 PL=0
MOVL C01170 V=800.0 PL=0
MOVL C01171 V=800.0 PL=0
MOVL C01172 V=800.0 PL=0
MOVL C01173 V=800.0 PL=0
MOVL C01174 V=800.0 PL=0
MOVL C01175 V=800.0 PL=0
MOVL C01176 V=800.0 PL=0
MOVL C01177 V=800.0 PL=0
MOVL C01178 V=800.0 PL=0
MOVL C01179 V=800.0 PL=0
MOVL C01180 V=800.0 PL=0
MOVL C01181 V=800.0 PL=0
MOVL C01182 V=800.0 PL=0
MOVL C01183 V=800.0 PL=0
MOVL C01184 V=800.0 PL=0
MOVL C01185 V=800.0 PL=0
MOVL C01186 V=800.0 PL=0
MOVL C01187 V=800.0 PL=0
MOVL C01188 V=800.0 PL=0
MOVL C01189 V=800.0 PL=0
MOVL C01190 V=800.0 PL=0
MOVL C01191 V=800.0 PL=0
MOVL C01192 V=800.0 PL=0
MOVL C01193 V=800.0 PL=0
MOVL C01194 V=800.0 PL=0
MOVL C01195 V=800.0 PL=0
MOVL C01196 V=800.0 PL=0
MOVL C01197 V=800.0 PL=0
MOVL C01198 V=800.0 PL=0
MOVL C01199 V=800.0 PL=0
MOVL C01200 V=800.0 PL=0
MOVL C01201 V=800.0 PL=0
MOVL C01202 V=800.0 PL=0
MOVL C01203 V=800.0 PL=0
MOVL C01204 V=800.0 PL=0
MOVL C01205 V=800.0 PL=0
MOVL C01206 V=800.0 PL=0
MOVL C01207 V=800.0 PL=0
MOVL C01208 V=800.0 PL=0
MOVL C01209 V=800.0 PL=0
MOVL C01210 V=800.0 PL=0
MOVL C01211 V=800.0 PL=0
MOVL C01212 V=800.0 PL=0
MOVL C01213 V=800.0 PL=0
MOVL C01214 V=800.0 PL=0
MOVL C01215 V=800.0 PL=0
MOVL C01216 V=800.0 PL=0
MOVL C01217 V=800.0 PL=0
MOVL C01218 V=800.0 PL=0
MOVL C01219 V=800.0 PL=0
MOVL C01220 V=800.0 PL=0
MOVL C01221 V=800.0 PL=0
MOVL C01222 V=800.0 PL=0
MOVL C01223 V=800.0 PL=0
MOVL C01224 V=800.0 PL=0
MOVL C01225 V=800.0 PL=0
MOVL C01226 V=800.0 PL=0
MOVL C01227 V=800.0 PL=0
MOVL C01228 V=800.0 PL=0
MOVL C01229 V=800.0 PL=0
MOVL C01230 V=800.0 PL=0
MOVL C01231 V=800.0 PL=0
MOVL C01232 V=800.0 PL=0
MOVL C01233 V=800.0 PL=0
MOVL C01234 V=800.0 PL=0
MOVL C01235 V=800.0 PL=0
MOVL C01236 V=800.0 PL=0
MOVL C01237 V=800.0 PL=0
MOVL C01238 V=800.0 PL=0
MOVL C01239 V=800.0 PL=0
MOVL C01240 V=800.0 PL=0
MOVL C01241 V=800.0 PL=0
MOVL C01242 V=800.0 PL=0
MOVL C01243 V=800.0 PL=0
MOVL C01244 V=800.0 PL=0
MOVL C01245 V=800.0 PL=0
MOVL C01246 V=800.0 PL=0
MOVL C01247 V=800.0 PL=0
MOVL C01248 V=800.0 PL=0
MOVL C01249 V=800.0 PL=0
MOVL C01250 V=800.0 PL=0
MOVL C01251 V=800.0 PL=0
MOVL C01252 V=800.0 PL=0
MOVL C01253 V=800.0 PL=0
MOVL C01254 V=800.0 PL=0
MOVL C01255 V=800.0 PL=0
MOVL C01256 V=800.0 PL=0
MOVL C01257 V=800.0 PL=0
MOVL C01258 V=800.0 PL=0
MOVL C01259 V=800.0 PL=0
MOVL C01260 V=800.0 PL=0
MOVL C01261 V=800.0 PL=0
MOVL C01262 V=800.0 PL=0
MOVL C01263 V=800.0 PL=0
MOVL C01264 V=800.0 PL=0
MOVL C01265 V=800.0 PL=0
MOVL C01266 V=800.0 PL=0
MOVL C01267 V=800.0 PL=0
MOVL C01268 V=800.0 PL=0
MOVL C01269 V=800.0 PL=0
MOVL C01270 V=800.0 PL=0
MOVL C01271 V=800.0 PL=0
MOVL C01272 V=800.0 PL=0
MOVL C01273 V=800.0 PL=0
MOVL C01274 V=800.0 PL=0
MOVL C01275 V=800.0 PL=0
MOVL C01276 V=800.0 PL=0
MOVL C01277 V=800.0 PL=0
MOVL C01278 V=800.0 PL=0
MOVL C01279 V=800.0 PL=0
MOVL C01280 V=800.0 PL=0
MOVL C01281 V=800.0 PL=0
MOVL C01282 V=800.0 PL=0
MOVL C01283 V=800.0 PL=0
MOVL C01284 V=800.0 PL=0
MOVL C01285 V=800.0 PL=0
MOVL C01286 V=800.0 PL=0
MOVL C01287 V=800.0 PL=0
MOVL C01288 V=800.0 PL=0
MOVL C01289 V=800.0 PL=0
MOVL C01290 V=800.0 PL=0
MOVL C01291 V=800.0 PL=0
MOVL C01292 V=800.0 PL=0
MOVL C01293 V=800.0 PL=0
MOVL C01294 V=800.0 PL=0
MOVL C01295 V=800.0 PL=0
MOVL C01296 V=800.0 PL=0
MOVL C01297 V=800.0 PL=0
MOVL C01298 V=800.0 PL=0
MOVL C01299 V=800.0 PL=0
MOVL C01300 V=800.0 PL=0
MOVL C01301 V=800.0 PL=0
MOVL C01302 V=800.0 PL=0
MOVL C01303 V=800.0 PL=0
MOVL C01304 V=800.0 PL=0
MOVL C01305 V=800.0 PL=0
MOVL C01306 V=800.0 PL=0
MOVL C01307 V=800.0 PL=0
MOVL C01308 V=800.0 PL=0
MOVL C01309 V=800.0 PL=0
MOVL C01310 V=800.0 PL=0
MOVL C01311 V=800.0 PL=0
MOVL C01312 V=800.0 PL=0
MOVL C01313 V=800.0 PL=0
MOVL C01314 V=800.0 PL=0
MOVL C01315 V=800.0 PL=0
MOVL C01316 V=800.0 PL=0
MOVL C01317 V=800.0 PL=0
MOVL C01318 V=800.0 PL=0
MOVL C01319 V=800.0 PL=0
MOVL C01320 V=800.0 PL=0
MOVL C01321 V=800.0 PL=0
MOVL C01322 V=800.0 PL=0
MOVL C01323 V=800.0 PL=0
MOVL C01324 V=800.0 PL=0
MOVL C01325 V=800.0 PL=0
MOVL C01326 V=800.0 PL=0
MOVL C01327 V=800.0 PL=0
MOVL C01328 V=800.0 PL=0
MOVL C01329 V=800.0 PL=0
MOVL C01330 V=800.0 PL=0
MOVL C01331 V=800.0 PL=0
MOVL C01332 V=800.0 PL=0
MOVL C01333 V=800.0 PL=0
MOVL C01334 V=800.0 PL=0
MOVL C01335 V=800.0 PL=0
MOVL C01336 V=800.0 PL=0
MOVL C01337 V=800.0 PL=0
MOVL C01338 V=800.0 PL=0
MOVL C01339 V=800.0 PL=0
MOVL C01340 V=800.0 PL=0
MOVL C01341 V=800.0 PL=0
MOVL C01342 V=800.0 PL=0
MOVL C01343 V=800.0 PL=0
MOVL C01344 V=800.0 PL=0
MOVL C01345 V=800.0 PL=0
MOVL C01346 V=800.0 PL=0
MOVL C01347 V=800.0 PL=0
MOVL C01348 V=800.0 PL=0
MOVL C01349 V=800.0 PL=0
MOVL C01350 V=800.0 PL=0
MOVL C01351 V=800.0 PL=0
MOVL C01352 V=800.0 PL=0
MOVL C01353 V=800.0 PL=0
MOVL C01354 V=800.0 PL=0
MOVL C01355 V=800.0 PL=0
MOVL C01356 V=800.0 PL=0
MOVL C01357 V=800.0 PL=0
MOVL C01358 V=800.0 PL=0
MOVL C01359 V=800.0 PL=0
MOVL C01360 V=800.0 PL=0
MOVL C01361 V=800.0 PL=0
MOVL C01362 V=800.0 PL=0
MOVL C01363 V=800.0 PL=0
MOVL C01364 V=800.0 PL=0
MOVL C01365 V=800.0 PL=0
MOVL C01366 V=800.0 PL=0
MOVL C01367 V=800.0 PL=0
MOVL C01368 V=800.0 PL=0
MOVL C01369 V=800.0 PL=0
MOVL C01370 V=800.0 PL=0
MOVL C01371 V=800.0 PL=0
MOVL C01372 V=800.0 PL=0
MOVL C01373 V=800.0 PL=0
MOVL C01374 V=800.0 PL=0
MOVL C01375 V=800.0 PL=0
MOVL C01376 V=800.0 PL=0
MOVL C01377 V=800.0 PL=0
MOVL C01378 V=800.0 PL=0
MOVL C01379 V=800.0 PL=0
MOVL C01380 V=800.0 PL=0
MOVL C01381 V=800.0 PL=0
MOVL C01382 V=800.0 PL=0
MOVL C01383 V=800.0 PL=0
MOVL C01384 V=800.0 PL=0
MOVL C01385 V=800.0 PL=0
MOVL C01386 V=800.0 PL=0
MOVL C01387 V=800.0 PL=0
MOVL C01388 V=800.0 PL=0
MOVL C01389 V=800.0 PL=0
MOVL C01390 V=800.0 PL=0
MOVL C01391 V=800.0 PL=0
MOVL C01392 V=800.0 PL=0
MOVL C01393 V=800.0 PL=0
MOVL C01394 V=800.0 PL=0
MOVL C01395 V=800.0 PL=0
MOVL C01396 V=800.0 PL=0
MOVL C01397 V=800.0 PL=0
MOVL C01398 V=800.0 PL=0
MOVL C01399 V=800.0 PL=0
MOVL C01400 V=800.0 PL=0
MOVL C01401 V=800.0 PL=0
MOVL C01402 V=800.0 PL=0
MOVL C01403 V=800.0 PL=0
MOVL C01404 V=800.0 PL=0
MOVL C01405 V=800.0 PL=0
MOVL C01406 V=800.0 PL=0
MOVL C01407 V=800.0 PL=0
MOVL C01408 V=800.0 PL=0
MOVL C01409 V=800.0 PL=0
MOVL C01410 V=800.0 PL=0
MOVL C01411 V=800.0 PL=0
MOVL C01412 V=800.0 PL=0
MOVL C01413 V=800.0 PL=0
MOVL C01414 V=800.0 PL=0
MOVL C01415 V=800.0 PL=0
MOVL C01416 V=800.0 PL=0
MOVL C01417 V=800.0 PL=0
MOVL C01418 V=800.0 PL=0
MOVL C01419 V=800.0 PL=0
MOVL C01420 V=800.0 PL=0
MOVL C01421 V=800.0 PL=0
MOVL C01422 V=800.0 PL=0
MOVL C01423 V=800.0 PL=0
MOVL C01424 V=800.0 PL=0
MOVL C01425 V=800.0 PL=0
MOVL C01426 V=800.0 PL=0
MOVL C01427 V=800.0 PL=0
MOVL C01428 V=800.0 PL=0
MOVL C01429 V=800.0 PL=0
MOVL C01430 V=800.0 PL=0
MOVL C01431 V=800.0 PL=0
MOVL C01432 V=800.0 PL=0
MOVL C01433 V=800.0 PL=0
MOVL C01434 V=800.0 PL=0
MOVL C01435 V=800.0 PL=0
MOVL C01436 V=800.0 PL=0
MOVL C01437 V=800.0 PL=0
MOVL C01438 V=800.0 PL=0
MOVL C01439 V=800.0 PL=0
MOVL C01440 V=800.0 PL=0
MOVL C01441 V=800.0 PL=0
MOVL C01442 V=800.0 PL=0
MOVL C01443 V=800.0 PL=0
MOVL C01444 V=800.0 PL=0
MOVL C01445 V=800.0 PL=0
MOVL C01446 V=800.0 PL=0
MOVL C01447 V=800.0 PL=0
MOVL C01448 V=800.0 PL=0
MOVL C01449 V=800.0 PL=0
MOVL C01450 V=800.0 PL=0
MOVL C01451 V=800.0 PL=0
MOVL C01452 V=800.0 PL=0
MOVL C01453 V=800.0 PL=0
MOVL C01454 V=800.0 PL=0
MOVL C01455 V=800.0 PL=0
MOVL C01456 V=800.0 PL=0
MOVL C01457 V=800.0 PL=0
MOVL C01458 V=800.0 PL=0
MOVL C01459 V=800.0 PL=0
MOVL C01460 V=800.0 PL=0
MOVL C01461 V=800.0 PL=0
MOVL C01462 V=800.0 PL=0
MOVL C01463 V=800.0 PL=0
MOVL C01464 V=800.0 PL=0
MOVL C01465 V=800.0 PL=0
MOVL C01466 V=800.0 PL=0
MOVL C01467 V=800.0 PL=0
MOVL C01468 V=800.0 PL=0
MOVL C01469 V=800.0 PL=0
MOVL C01470 V=800.0 PL=0
MOVL C01471 V=800.0 PL=0
MOVL C01472 V=800.0 PL=0
MOVL C01473 V=800.0 PL=0
MOVL C01474 V=800.0 PL=0
MOVL C01475 V=800.0 PL=0
MOVL C01476 V=800.0 PL=0
MOVL C01477 V=800.0 PL=0
MOVL C01478 V=800.0 PL=0
MOVL C01479 V=800.0 PL=0
MOVL C01480 V=800.0 PL=0
MOVL C01481 V=800.0 PL=0
MOVL C01482 V=800.0 PL=0
MOVL C01483 V=800.0 PL=0
MOVL C01484 V=800.0 PL=0
MOVL C01485 V=800.0 PL=0
MOVL C01486 V=800.0 PL=0
MOVL C01487 V=800.0 PL=0
MOVL C01488 V=800.0 PL=0
MOVL C01489 V=800.0 PL=0
MOVL C01490 V=800.0 PL=0
MOVL C01491 V=800.0 PL=0
MOVL C01492 V=800.0 PL=0
MOVL C01493 V=800.0 PL=0
MOVL C01494 V=800.0 PL=0
MOVL C01495 V=800.0 PL=0
MOVL C01496 V=800.0 PL=0
MOVL C01497 V=800.0 PL=0
MOVL C01498 V=800.0 PL=0
MOVL C01499 V=800.0 PL=0
MOVL C01500 V=800.0 PL=0
MOVL C01501 V=800.0 PL=0
MOVL C01502 V=800.0 PL=0
MOVL C01503 V=800.0 PL=0
MOVL C01504 V=800.0 PL=0
MOVL C01505 V=800.0 PL=0
MOVL C01506 V=800.0 PL=0
MOVL C01507 V=800.0 PL=0
MOVL C01508 V=800.0 PL=0
MOVL C01509 V=800.0 PL=0
MOVL C01510 V=800.0 PL=0
MOVL C01511 V=800.0 PL=0
MOVL C01512 V=800.0 PL=0
MOVL C01513 V=800.0 PL=0
MOVL C01514 V=800.0 PL=0
MOVL C01515 V=800.0 PL=0
MOVL C01516 V=800.0 PL=0
MOVL C01517 V=800.0 PL=0
MOVL C01518 V=800.0 PL=0
MOVL C01519 V=800.0 PL=0
MOVL C01520 V=800.0 PL=0
MOVL C01521 V=800.0 PL=0
MOVL C01522 V=800.0 PL=0
MOVL C01523 V=800.0 PL=0
MOVL C01524 V=800.0 PL=0
MOVL C01525 V=800.0 PL=0
MOVL C01526 V=800.0 PL=0
MOVL C01527 V=800.0 PL=0
MOVL C01528 V=800.0 PL=0
MOVL C01529 V=800.0 PL=0
MOVL C01530 V=800.0 PL=0
MOVL C01531 V=800.0 PL=0
MOVL C01532 V=800.0 PL=0
MOVL C01533 V=800.0 PL=0
MOVL C01534 V=800.0 PL=0
MOVL C01535 V=800.0 PL=0
MOVL C01536 V=800.0 PL=0
MOVL C01537 V=800.0 PL=0
MOVL C01538 V=800.0 PL=0
MOVL C01539 V=800.0 PL=0
MOVL C01540 V=800.0 PL=0
MOVL C01541 V=800.0 PL=0
MOVL C01542 V=800.0 PL=0
MOVL C01543 V=800.0 PL=0
MOVL C01544 V=800.0 PL=0
MOVL C01545 V=800.0 PL=0
MOVL C01546 V=800.0 PL=0
MOVL C01547 V=800.0 PL=0
MOVL C01548 V=800.0 PL=0
MOVL C01549 V=800.0 PL=0
MOVL C01550 V=800.0 PL=0
MOVL C01551 V=800.0 PL=0
MOVL C01552 V=800.0 PL=0
MOVL C01553 V=800.0 PL=0
MOVL C01554 V=800.0 PL=0
MOVL C01555 V=800.0 PL=0
MOVL C01556 V=800.0 PL=0
MOVL C01557 V=800.0 PL=0
MOVL C01558 V=800.0 PL=0
MOVL C01559 V=800.0 PL=0
MOVL C01560 V=800.0 PL=0
MOVL C01561 V=800.0 PL=0
MOVL C01562 V=800.0 PL=0
MOVL C01563 V=800.0 PL=0
MOVL C01564 V=800.0 PL=0
MOVL C01565 V=800.0 PL=0
MOVL C01566 V=800.0 PL=0
MOVL C01567 V=800.0 PL=0
MOVL C01568 V=800.0 PL=0
MOVL C01569 V=800.0 PL=0
MOVL C01570 V=800.0 PL=0
MOVL C01571 V=800.0 PL=0
MOVL C01572 V=800.0 PL=0
MOVL C01573 V=800.0 PL=0
MOVL C01574 V=800.0 PL=0
MOVL C01575 V=800.0 PL=0
MOVL C01576 V=800.0 PL=0
MOVL C01577 V=800.0 PL=0
MOVL C01578 V=800.0 PL=0
MOVL C01579 V=800.0 PL=0
MOVL C01580 V=800.0 PL=0
MOVL C01581 V=800.0 PL=0
MOVL C01582 V=800.0 PL=0
MOVL C01583 V=800.0 PL=0
MOVL C01584 V=800.0 PL=0
MOVL C01585 V=800.0 PL=0
MOVL C01586 V=800.0 PL=0
MOVL C01587 V=800.0 PL=0
MOVL C01588 V=800.0 PL=0
MOVL C01589 V=800.0 PL=0
MOVL C01590 V=800.0 PL=0
MOVL C01591 V=800.0 PL=0
MOVL C01592 V=800.0 PL=0
MOVL C01593 V=800.0 PL=0
MOVL C01594 V=800.0 PL=0
MOVL C01595 V=800.0 PL=0
MOVL C01596 V=800.0 PL=0
MOVL C01597 V=800.0 PL=0
MOVL C01598 V=800.0 PL=0
MOVL C01599 V=800.0 PL=0
MOVL C01600 V=800.0 PL=0
MOVL C01601 V=800.0 PL=0
MOVL C01602 V=800.0 PL=0
MOVL C01603 V=800.0 PL=0
MOVL C01604 V=800.0 PL=0
MOVL C01605 V=800.0 PL=0
MOVL C01606 V=800.0 PL=0
MOVL C01607 V=800.0 PL=0
MOVL C01608 V=800.0 PL=0
MOVL C01609 V=800.0 PL=0
MOVL C01610 V=800.0 PL=0
MOVL C01611 V=800.0 PL=0
MOVL C01612 V=800.0 PL=0
MOVL C01613 V=800.0 PL=0
MOVL C01614 V=800.0 PL=0
MOVL C01615 V=800.0 PL=0
MOVL C01616 V=800.0 PL=0
MOVL C01617 V=800.0 PL=0
MOVL C01618 V=800.0 PL=0
MOVL C01619 V=800.0 PL=0
MOVL C01620 V=800.0 PL=0
MOVL C01621 V=800.0 PL=0
MOVL C01622 V=800.0 PL=0
MOVL C01623 V=800.0 PL=0
MOVL C01624 V=800.0 PL=0
MOVL C01625 V=800.0 PL=0
MOVL C01626 V=800.0 PL=0
MOVL C01627 V=800.0 PL=0
MOVL C01628 V=800.0 PL=0
MOVL C01629 V=800.0 PL=0
MOVL C01630 V=800.0 PL=0
MOVL C01631 V=800.0 PL=0
MOVL C01632 V=800.0 PL=0
MOVL C01633 V=800.0 PL=0
MOVL C01634 V=800.0 PL=0
MOVL C01635 V=800.0 PL=0
MOVL C01636 V=800.0 PL=0
MOVL C01637 V=800.0 PL=0
MOVL C01638 V=800.0 PL=0
MOVL C01639 V=800.0 PL=0
MOVL C01640 V=800.0 PL=0
MOVL C01641 V=800.0 PL=0
MOVL C01642 V=800.0 PL=0
MOVL C01643 V=800.0 PL=0
MOVL C01644 V=800.0 PL=0
MOVL C01645 V=800.0 PL=0
MOVL C01646 V=800.0 PL=0
MOVL C01647 V=800.0 PL=0
MOVL C01648 V=800.0 PL=0
MOVL C01649 V=800.0 PL=0
MOVL C01650 V=800.0 PL=0
MOVL C01651 V=800.0 PL=0
MOVL C01652 V=800.0 PL=0
MOVL C01653 V=800.0 PL=0
MOVL C01654 V=800.0 PL=0
MOVL C01655 V=800.0 PL=0
MOVL C01656 V=800.0 PL=0
MOVL C01657 V=800.0 PL=0
MOVL C01658 V=800.0 PL=0
MOVL C01659 V=800.0 PL=0
MOVL C01660 V=800.0 PL=0
MOVL C01661 V=800.0 PL=0
MOVL C01662 V=800.0 PL=0
MOVL C01663 V=800.0 PL=0
MOVL C01664 V=800.0 PL=0
MOVL C01665 V=800.0 PL=0
MOVL C01666 V=800.0 PL=0
MOVL C01667 V=800.0 PL=0
MOVL C01668 V=800.0 PL=0
MOVL C01669 V=800.0 PL=0
MOVL C01670 V=800.0 PL=0
MOVL C01671 V=800.0 PL=0
MOVL C01672 V=800.0 PL=0
MOVL C01673 V=800.0 PL=0
MOVL C01674 V=800.0 PL=0
MOVL C01675 V=800.0 PL=0
MOVL C01676 V=800.0 PL=0
MOVL C01677 V=800.0 PL=0
MOVL C01678 V=800.0 PL=0
MOVL C01679 V=800.0 PL=0
MOVL C01680 V=800.0 PL=0
MOVL C01681 V=800.0 PL=0
MOVL C01682 V=800.0 PL=0
MOVL C01683 V=800.0 PL=0
MOVL C01684 V=800.0 PL=0
MOVL C01685 V=800.0 PL=0
MOVL C01686 V=800.0 PL=0
MOVL C01687 V=800.0 PL=0
MOVL C01688 V=800.0 PL=0
MOVL C01689 V=800.0 PL=0
MOVL C01690 V=800.0 PL=0
MOVL C01691 V=800.0 PL=0
MOVL C01692 V=800.0 PL=0
MOVL C01693 V=800.0 PL=0
MOVL C01694 V=800.0 PL=0
MOVL C01695 V=800.0 PL=0
MOVL C01696 V=800.0 PL=0
MOVL C01697 V=800.0 PL=0
MOVL C01698 V=800.0 PL=0
MOVL C01699 V=800.0 PL=0
MOVL C01700 V=800.0 PL=0
MOVL C01701 V=800.0 PL=0
MOVL C01702 V=800.0 PL=0
MOVL C01703 V=800.0 PL=0
MOVL C01704 V=800.0 PL=0
MOVL C01705 V=800.0 PL=0
MOVL C01706 V=800.0 PL=0
MOVL C01707 V=800.0 PL=0
MOVL C01708 V=800.0 PL=0
MOVL C01709 V=800.0 PL=0
MOVL C01710 V=800.0 PL=0
MOVL C01711 V=800.0 PL=0
MOVL C01712 V=800.0 PL=0
MOVL C01713 V=800.0 PL=0
MOVL C01714 V=800.0 PL=0
MOVL C01715 V=800.0 PL=0
MOVL C01716 V=800.0 PL=0
MOVL C01717 V=800.0 PL=0
MOVL C01718 V=800.0 PL=0
MOVL C01719 V=800.0 PL=0
MOVL C01720 V=800.0 PL=0
MOVL C01721 V=800.0 PL=0
MOVL C01722 V=800.0 PL=0
MOVL C01723 V=800.0 PL=0
MOVL C01724 V=800.0 PL=0
MOVL C01725 V=800.0 PL=0
MOVL C01726 V=800.0 PL=0
MOVL C01727 V=800.0 PL=0
MOVL C01728 V=800.0 PL=0
MOVL C01729 V=800.0 PL=0
MOVL C01730 V=800.0 PL=0
MOVL C01731 V=800.0 PL=0
MOVL C01732 V=800.0 PL=0
MOVL C01733 V=800.0 PL=0
MOVL C01734 V=800.0 PL=0
MOVL C01735 V=800.0 PL=0
MOVL C01736 V=800.0 PL=0
MOVL C01737 V=800.0 PL=0
MOVL C01738 V=800.0 PL=0
MOVL C01739 V=800.0 PL=0
MOVL C01740 V=800.0 PL=0
MOVL C01741 V=800.0 PL=0
MOVL C01742 V=800.0 PL=0
MOVL C01743 V=800.0 PL=0
MOVL C01744 V=800.0 PL=0
MOVL C01745 V=800.0 PL=0
MOVL C01746 V=800.0 PL=0
MOVL C01747 V=800.0 PL=0
MOVL C01748 V=800.0 PL=0
MOVL C01749 V=800.0 PL=0
MOVL C01750 V=800.0 PL=0
MOVL C01751 V=800.0 PL=0
MOVL C01752 V=800.0 PL=0
MOVL C01753 V=800.0 PL=0
MOVL C01754 V=800.0 PL=0
MOVL C01755 V=800.0 PL=0
MOVL C01756 V=800.0 PL=0
MOVL C01757 V=800.0 PL=0
MOVL C01758 V=800.0 PL=0
MOVL C01759 V=800.0 PL=0
MOVL C01760 V=800.0 PL=0
MOVL C01761 V=800.0 PL=0
MOVL C01762 V=800.0 PL=0
MOVL C01763 V=800.0 PL=0
MOVL C01764 V=800.0 PL=0
MOVL C01765 V=800.0 PL=0
MOVL C01766 V=800.0 PL=0
MOVL C01767 V=800.0 PL=0
MOVL C01768 V=800.0 PL=0
MOVL C01769 V=800.0 PL=0
MOVL C01770 V=800.0 PL=0
MOVL C01771 V=800.0 PL=0
MOVL C01772 V=800.0 PL=0
MOVL C01773 V=800.0 PL=0
MOVL C01774 V=800.0 PL=0
MOVL C01775 V=800.0 PL=0
MOVL C01776 V=800.0 PL=0
MOVL C01777 V=800.0 PL=0
MOVL C01778 V=800.0 PL=0
MOVL C01779 V=800.0 PL=0
MOVL C01780 V=800.0 PL=0
MOVL C01781 V=800.0 PL=0
MOVL C01782 V=800.0 PL=0
MOVL C01783 V=800.0 PL=0
MOVL C01784 V=800.0 PL=0
MOVL C01785 V=800.0 PL=0
MOVL C01786 V=800.0 PL=0
MOVL C01787 V=800.0 PL=0
MOVL C01788 V=800.0 PL=0
MOVL C01789 V=800.0 PL=0
MOVL C01790 V=800.0 PL=0
MOVL C01791 V=800.0 PL=0
MOVL C01792 V=800.0 PL=0
MOVL C01793 V=800.0 PL=0
MOVL C01794 V=800.0 PL=0
MOVL C01795 V=800.0 PL=0
MOVL C01796 V=800.0 PL=0
MOVL C01797 V=800.0 PL=0
MOVL C01798 V=800.0 PL=0
MOVL C01799 V=800.0 PL=0
MOVL C01800 V=800.0 PL=0
MOVL C01801 V=800.0 PL=0
MOVL C01802 V=800.0 PL=0
MOVL C01803 V=800.0 PL=0
MOVL C01804 V=800.0 PL=0
MOVL C01805 V=800.0 PL=0
MOVL C01806 V=800.0 PL=0
MOVL C01807 V=800.0 PL=0
MOVL C01808 V=800.0 PL=0
MOVL C01809 V=800.0 PL=0
MOVL C01810 V=800.0 PL=0
MOVL C01811 V=800.0 PL=0
MOVL C01812 V=800.0 PL=0
MOVL C01813 V=800.0 PL=0
MOVL C01814 V=800.0 PL=0
MOVL C01815 V=800.0 PL=0
MOVL C01816 V=800.0 PL=0
MOVL C01817 V=800.0 PL=0
MOVL C01818 V=800.0 PL=0
MOVL C01819 V=800.0 PL=0
MOVL C01820 V=800.0 PL=0
MOVL C01821 V=800.0 PL=0
MOVL C01822 V=800.0 PL=0
MOVL C01823 V=800.0 PL=0
MOVL C01824 V=800.0 PL=0
MOVL C01825 V=800.0 PL=0
MOVL C01826 V=800.0 PL=0
MOVL C01827 V=800.0 PL=0
MOVL C01828 V=800.0 PL=0
MOVL C01829 V=800.0 PL=0
MOVL C01830 V=800.0 PL=0
MOVL C01831 V=800.0 PL=0
MOVL C01832 V=800.0 PL=0
MOVL C01833 V=800.0 PL=0
MOVL C01834 V=800.0 PL=0
MOVL C01835 V=800.0 PL=0
MOVL C01836 V=800.0 PL=0
MOVL C01837 V=800.0 PL=0
MOVL C01838 V=800.0 PL=0
MOVL C01839 V=800.0 PL=0
MOVL C01840 V=800.0 PL=0
MOVL C01841 V=800.0 PL=0
MOVL C01842 V=800.0 PL=0
MOVL C01843 V=800.0 PL=0
MOVL C01844 V=800.0 PL=0
MOVL C01845 V=800.0 PL=0
MOVL C01846 V=800.0 PL=0
MOVL C01847 V=800.0 PL=0
MOVL C01848 V=800.0 PL=0
MOVL C01849 V=800.0 PL=0
MOVL C01850 V=800.0 PL=0
MOVL C01851 V=800.0 PL=0
MOVL C01852 V=800.0 PL=0
MOVL C01853 V=800.0 PL=0
MOVL C01854 V=800.0 PL=0
MOVL C01855 V=800.0 PL=0
MOVL C01856 V=800.0 PL=0
MOVL C01857 V=800.0 PL=0
MOVL C01858 V=800.0 PL=0
MOVL C01859 V=800.0 PL=0
MOVL C01860 V=800.0 PL=0
MOVL C01861 V=800.0 PL=0
MOVL C01862 V=800.0 PL=0
MOVL C01863 V=800.0 PL=0
MOVL C01864 V=800.0 PL=0
MOVL C01865 V=800.0 PL=0
MOVL C01866 V=800.0 PL=0
MOVL C01867 V=800.0 PL=0
MOVL C01868 V=800.0 PL=0
MOVL C01869 V=800.0 PL=0
MOVL C01870 V=800.0 PL=0
MOVL C01871 V=800.0 PL=0
MOVL C01872 V=800.0 PL=0
MOVL C01873 V=800.0 PL=0
MOVL C01874 V=800.0 PL=0
MOVL C01875 V=800.0 PL=0
MOVL C01876 V=800.0 PL=0
MOVL C01877 V=800.0 PL=0
MOVL C01878 V=800.0 PL=0
MOVL C01879 V=800.0 PL=0
MOVL C01880 V=800.0 PL=0
MOVL C01881 V=800.0 PL=0
MOVL C01882 V=800.0 PL=0
MOVL C01883 V=800.0 PL=0
MOVL C01884 V=800.0 PL=0
MOVL C01885 V=800.0 PL=0
MOVL C01886 V=800.0 PL=0
MOVL C01887 V=800.0 PL=0
MOVL C01888 V=800.0 PL=0
MOVL C01889 V=800.0 PL=0
MOVL C01890 V=800.0 PL=0
MOVL C01891 V=800.0 PL=0
MOVL C01892 V=800.0 PL=0
MOVL C01893 V=800.0 PL=0
MOVL C01894 V=800.0 PL=0
MOVL C01895 V=800.0 PL=0
MOVL C01896 V=800.0 PL=0
MOVL C01897 V=800.0 PL=0
MOVL C01898 V=800.0 PL=0
MOVL C01899 V=800.0 PL=0
MOVL C01900 V=800.0 PL=0
MOVL C01901 V=800.0 PL=0
MOVL C01902 V=800.0 PL=0
MOVL C01903 V=800.0 PL=0
MOVL C01904 V=800.0 PL=0
MOVL C01905 V=800.0 PL=0
MOVL C01906 V=800.0 PL=0
MOVL C01907 V=800.0 PL=0
MOVL C01908 V=800.0 PL=0
MOVL C01909 V=800.0 PL=0
MOVL C01910 V=800.0 PL=0
MOVL C01911 V=800.0 PL=0
MOVL C01912 V=800.0 PL=0
MOVL C01913 V=800.0 PL=0
MOVL C01914 V=800.0 PL=0
MOVL C01915 V=800.0 PL=0
MOVL C01916 V=800.0 PL=0
MOVL C01917 V=800.0 PL=0
MOVL C01918 V=800.0 PL=0
MOVL C01919 V=800.0 PL=0
MOVL C01920 V=800.0 PL=0
MOVL C01921 V=800.0 PL=0
MOVL C01922 V=800.0 PL=0
MOVL C01923 V=800.0 PL=0
MOVL C01924 V=800.0 PL=0
MOVL C01925 V=800.0 PL=0
MOVL C01926 V=800.0 PL=0
MOVL C01927 V=800.0 PL=0
MOVL C01928 V=800.0 PL=0
MOVL C01929 V=800.0 PL=0
MOVL C01930 V=800.0 PL=0
MOVL C01931 V=800.0 PL=0
MOVL C01932 V=800.0 PL=0
MOVL C01933 V=800.0 PL=0
MOVL C01934 V=800.0 PL=0
MOVL C01935 V=800.0 PL=0
MOVL C01936 V=800.0 PL=0
MOVL C01937 V=800.0 PL=0
MOVL C01938 V=800.0 PL=0
MOVL C01939 V=800.0 PL=0
MOVL C01940 V=800.0 PL=0
MOVL C01941 V=800.0 PL=0
MOVL C01942 V=800.0 PL=0
MOVL C01943 V=800.0 PL=0
MOVL C01944 V=800.0 PL=0
MOVL C01945 V=800.0 PL=0
MOVL C01946 V=800.0 PL=0
MOVL C01947 V=800.0 PL=0
MOVL C01948 V=800.0 PL=0
MOVL C01949 V=800.0 PL=0
MOVL C01950 V=800.0 PL=0
MOVL C01951 V=800.0 PL=0
MOVL C01952 V=800.0 PL=0
MOVL C01953 V=800.0 PL=0
MOVL C01954 V=800.0 PL=0
MOVL C01955 V=800.0 PL=0
MOVL C01956 V=800.0 PL=0
MOVL C01957 V=800.0 PL=0
MOVL C01958 V=800.0 PL=0
MOVL C01959 V=800.0 PL=0
MOVL C01960 V=800.0 PL=0
MOVL C01961 V=800.0 PL=0
MOVL C01962 V=800.0 PL=0
MOVL C01963 V=800.0 PL=0
MOVL C01964 V=800.0 PL=0
MOVL C01965 V=800.0 PL=0
MOVL C01966 V=800.0 PL=0
MOVL C01967 V=800.0 PL=0
MOVL C01968 V=800.0 PL=0
MOVL C01969 V=800.0 PL=0
MOVL C01970 V=800.0 PL=0
MOVL C01971 V=800.0 PL=0
MOVL C01972 V=800.0 PL=0
MOVL C01973 V=800.0 PL=0
